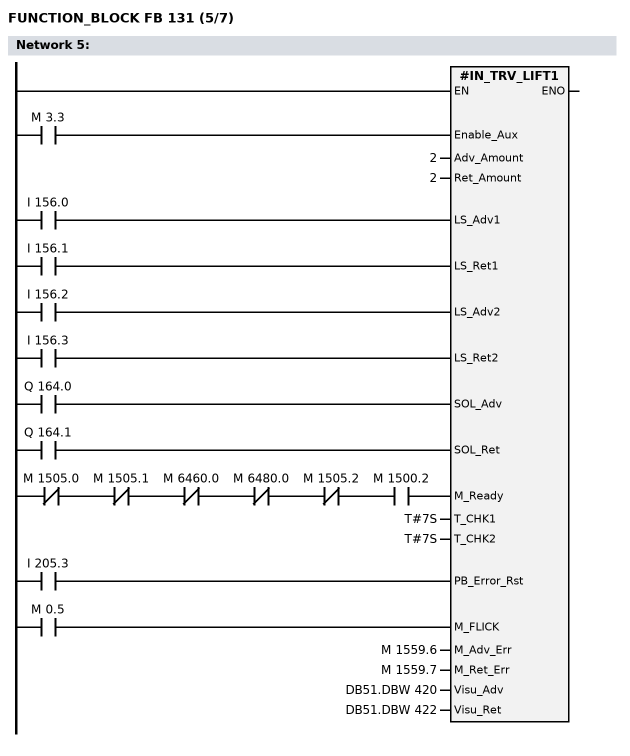

      A     M      3.3;
      =     L      0.0;
      BLD   103;
      A     I    156.0;
      =     L      0.1;
      BLD   103;
      A     I    156.1;
      =     L      0.2;
      BLD   103;
      A     I    156.2;
      =     L      0.3;
      BLD   103;
      A     I    156.3;
      =     L      0.4;
      BLD   103;
      A     Q    164.0;
      =     L      1.1;
      BLD   103;
      A     Q    164.1;
      =     L      1.2;
      BLD   103;
      AN    M   1505.0;
      AN    M   1505.1;
      AN    M   6460.0;
      AN    M   6480.0;
      AN    M   1505.2;
      A     M   1500.2;
      =     L      1.3;
      BLD   103;
      A     I    205.3;
      =     L      1.5;
      BLD   103;
      A     M      0.5;
      =     L      1.6;
      BLD   103;
      CALL #IN_TRV_LIFT1 (
           Enable_Aux               := L      0.0,
           Adv_Amount               := 2,
           Ret_Amount               := 2,
           LS_Adv1                  := L      0.1,
           LS_Ret1                  := L      0.2,
           LS_Adv2                  := L      0.3,
           LS_Ret2                  := L      0.4,
           SOL_Adv                  := L      1.1,
           SOL_Ret                  := L      1.2,
           M_Ready                  := L      1.3,
           T_CHK1                   := T#7S,
           T_CHK2                   := T#7S,
           PB_Error_Rst             := L      1.5,
           M_FLICK                  := L      1.6,
           M_Adv_Err                := M   1559.6,
           M_Ret_Err                := M   1559.7,
           Visu_Adv                 := DB51.DBW  420,
           Visu_Ret                 := DB51.DBW  422);
      NOP   0;
NETWORK
TITLE =
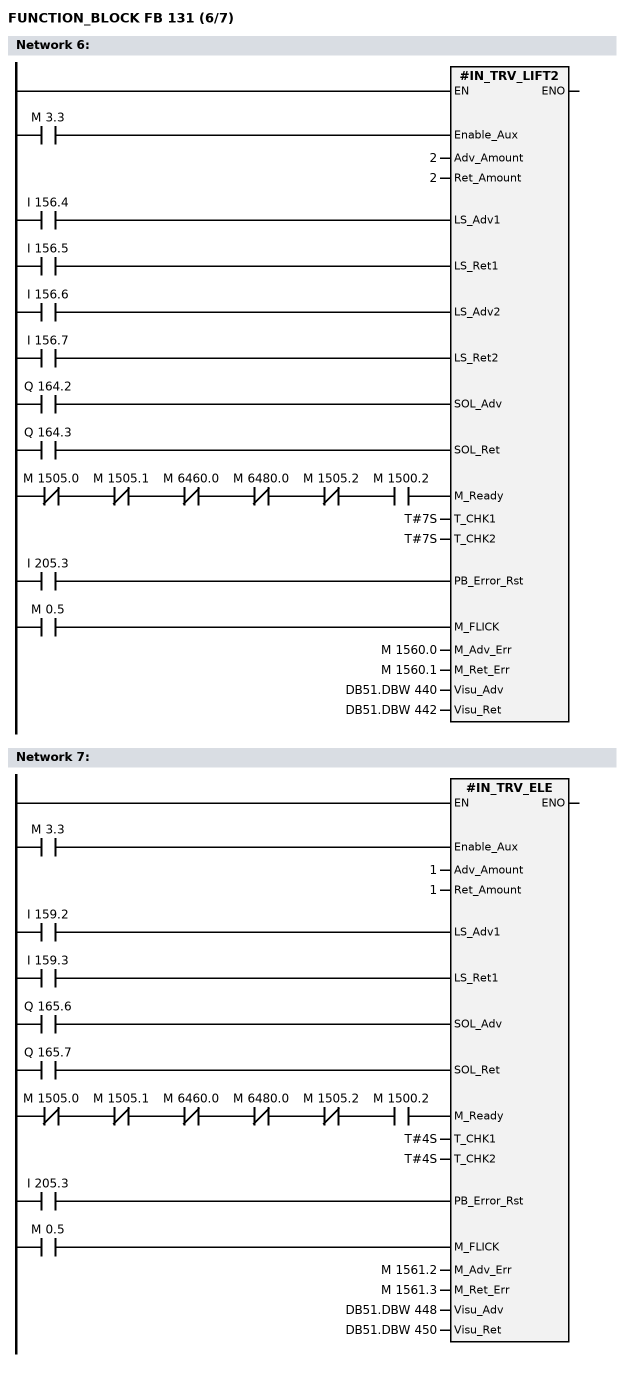

      A     M      3.3;
      =     L      0.0;
      BLD   103;
      A     I    156.4;
      =     L      0.1;
      BLD   103;
      A     I    156.5;
      =     L      0.2;
      BLD   103;
      A     I    156.6;
      =     L      0.3;
      BLD   103;
      A     I    156.7;
      =     L      0.4;
      BLD   103;
      A     Q    164.2;
      =     L      1.1;
      BLD   103;
      A     Q    164.3;
      =     L      1.2;
      BLD   103;
      AN    M   1505.0;
      AN    M   1505.1;
      AN    M   6460.0;
      AN    M   6480.0;
      AN    M   1505.2;
      A     M   1500.2;
      =     L      1.3;
      BLD   103;
      A     I    205.3;
      =     L      1.5;
      BLD   103;
      A     M      0.5;
      =     L      1.6;
      BLD   103;
      CALL #IN_TRV_LIFT2 (
           Enable_Aux               := L      0.0,
           Adv_Amount               := 2,
           Ret_Amount               := 2,
           LS_Adv1                  := L      0.1,
           LS_Ret1                  := L      0.2,
           LS_Adv2                  := L      0.3,
           LS_Ret2                  := L      0.4,
           SOL_Adv                  := L      1.1,
           SOL_Ret                  := L      1.2,
           M_Ready                  := L      1.3,
           T_CHK1                   := T#7S,
           T_CHK2                   := T#7S,
           PB_Error_Rst             := L      1.5,
           M_FLICK                  := L      1.6,
           M_Adv_Err                := M   1560.0,
           M_Ret_Err                := M   1560.1,
           Visu_Adv                 := DB51.DBW  440,
           Visu_Ret                 := DB51.DBW  442);
      NOP   0;
NETWORK
TITLE =

      A     M      3.3;
      =     L      0.0;
      BLD   103;
      A     I    159.2;
      =     L      0.1;
      BLD   103;
      A     I    159.3;
      =     L      0.2;
      BLD   103;
      A     Q    165.6;
      =     L      1.1;
      BLD   103;
      A     Q    165.7;
      =     L      1.2;
      BLD   103;
      AN    M   1505.0;
      AN    M   1505.1;
      AN    M   6460.0;
      AN    M   6480.0;
      AN    M   1505.2;
      A     M   1500.2;
      =     L      1.3;
      BLD   103;
      A     I    205.3;
      =     L      1.5;
      BLD   103;
      A     M      0.5;
      =     L      1.6;
      BLD   103;
      CALL #IN_TRV_ELE (
           Enable_Aux               := L      0.0,
           Adv_Amount               := 1,
           Ret_Amount               := 1,
           LS_Adv1                  := L      0.1,
           LS_Ret1                  := L      0.2,
           SOL_Adv                  := L      1.1,
           SOL_Ret                  := L      1.2,
           M_Ready                  := L      1.3,
           T_CHK1                   := T#4S,
           T_CHK2                   := T#4S,
           PB_Error_Rst             := L      1.5,
           M_FLICK                  := L      1.6,
           M_Adv_Err                := M   1561.2,
           M_Ret_Err                := M   1561.3,
           Visu_Adv                 := DB51.DBW  448,
           Visu_Ret                 := DB51.DBW  450);
      NOP   0;
NETWORK
TITLE =
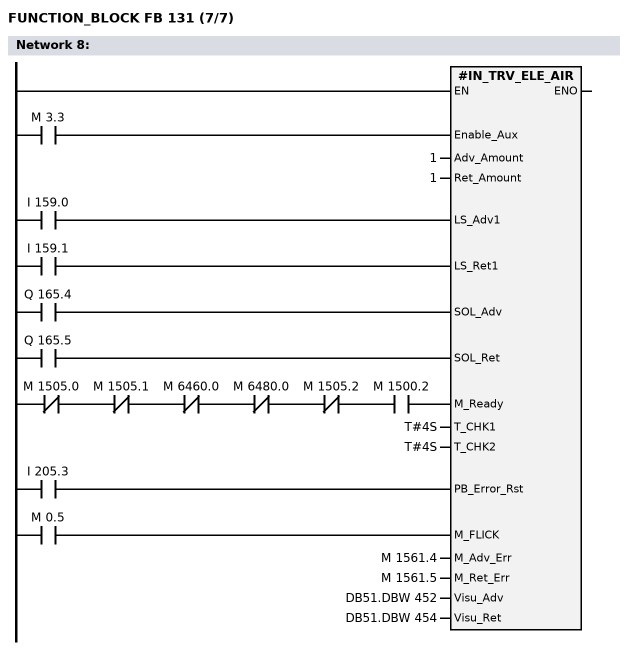

      A     M      3.3;
      =     L      0.0;
      BLD   103;
      A     I    159.0;
      =     L      0.1;
      BLD   103;
      A     I    159.1;
      =     L      0.2;
      BLD   103;
      A     Q    165.4;
      =     L      1.1;
      BLD   103;
      A     Q    165.5;
      =     L      1.2;
      BLD   103;
      AN    M   1505.0;
      AN    M   1505.1;
      AN    M   6460.0;
      AN    M   6480.0;
      AN    M   1505.2;
      A     M   1500.2;
      =     L      1.3;
      BLD   103;
      A     I    205.3;
      =     L      1.5;
      BLD   103;
      A     M      0.5;
      =     L      1.6;
      BLD   103;
      CALL #IN_TRV_ELE_AIR (
           Enable_Aux               := L      0.0,
           Adv_Amount               := 1,
           Ret_Amount               := 1,
           LS_Adv1                  := L      0.1,
           LS_Ret1                  := L      0.2,
           SOL_Adv                  := L      1.1,
           SOL_Ret                  := L      1.2,
           M_Ready                  := L      1.3,
           T_CHK1                   := T#4S,
           T_CHK2                   := T#4S,
           PB_Error_Rst             := L      1.5,
           M_FLICK                  := L      1.6,
           M_Adv_Err                := M   1561.4,
           M_Ret_Err                := M   1561.5,
           Visu_Adv                 := DB51.DBW  452,
           Visu_Ret                 := DB51.DBW  454);
      NOP   0;
END_FUNCTION_BLOCK

DATA_BLOCK DB 131
TITLE =
VERSION : 0.0

 FB 131
BEGIN
   IN_TRV_CUSHION_B.Enable_Aux := FALSE;
   IN_TRV_CUSHION_B.Adv_Amount := 0;
   IN_TRV_CUSHION_B.Ret_Amount := 0;
   IN_TRV_CUSHION_B.LS_Adv1 := FALSE;
   IN_TRV_CUSHION_B.LS_Ret1 := FALSE;
   IN_TRV_CUSHION_B.LS_Adv2 := FALSE;
   IN_TRV_CUSHION_B.LS_Ret2 := FALSE;
   IN_TRV_CUSHION_B.LS_Adv3 := FALSE;
   IN_TRV_CUSHION_B.LS_Ret3 := FALSE;
   IN_TRV_CUSHION_B.LS_Adv4 := FALSE;
   IN_TRV_CUSHION_B.LS_Ret4 := FALSE;
   IN_TRV_CUSHION_B.SOL_Adv := FALSE;
   IN_TRV_CUSHION_B.SOL_Ret := FALSE;
   IN_TRV_CUSHION_B.M_Ready := FALSE;
   IN_TRV_CUSHION_B.T_CHK1 := T#0MS;
   IN_TRV_CUSHION_B.T_CHK2 := T#0MS;
   IN_TRV_CUSHION_B.PB_Lamp_CHK := FALSE;
   IN_TRV_CUSHION_B.PB_Error_Rst := FALSE;
   IN_TRV_CUSHION_B.M_FLICK := FALSE;
   IN_TRV_CUSHION_B.M_Adv_Err := FALSE;
   IN_TRV_CUSHION_B.M_Ret_Err := FALSE;
   IN_TRV_CUSHION_B.LP_Adv := FALSE;
   IN_TRV_CUSHION_B.LP_Ret := FALSE;
   IN_TRV_CUSHION_B.Visu_Adv := W#16#0;
   IN_TRV_CUSHION_B.Visu_Ret := W#16#0;
   IN_TRV_CUSHION_B.Error_T1.IN := FALSE;
   IN_TRV_CUSHION_B.Error_T1.PT := T#0MS;
   IN_TRV_CUSHION_B.Error_T1.Q := FALSE;
   IN_TRV_CUSHION_B.Error_T1.ET := T#0MS;
   IN_TRV_CUSHION_B.Error_T1.STATE := B#16#0;
   IN_TRV_CUSHION_B.Error_T1.STIME := T#0MS;
   IN_TRV_CUSHION_B.Error_T1.ATIME := T#0MS;
   IN_TRV_CUSHION_B.Error_T2.IN := FALSE;
   IN_TRV_CUSHION_B.Error_T2.PT := T#0MS;
   IN_TRV_CUSHION_B.Error_T2.Q := FALSE;
   IN_TRV_CUSHION_B.Error_T2.ET := T#0MS;
   IN_TRV_CUSHION_B.Error_T2.STATE := B#16#0;
   IN_TRV_CUSHION_B.Error_T2.STIME := T#0MS;
   IN_TRV_CUSHION_B.Error_T2.ATIME := T#0MS;
   IN_TRV_CUSHION_B.CHK_Aux1 := FALSE;
   IN_TRV_CUSHION_B.CHK_Aux2 := FALSE;
   IN_TRV_CUSHION_B.Error_T1_DN := FALSE;
   IN_TRV_CUSHION_B.Error_T2_DN := FALSE;
   IN_TRV_CUSHION_B.Adv_Memo := FALSE;
   IN_TRV_CUSHION_B.Visu_Adv_Arr[0] := FALSE;
   IN_TRV_CUSHION_B.Visu_Adv_Arr[1] := FALSE;
   IN_TRV_CUSHION_B.Visu_Adv_Arr[2] := FALSE;
   IN_TRV_CUSHION_B.Visu_Adv_Arr[3] := FALSE;
   IN_TRV_CUSHION_B.Visu_Adv_Arr[4] := FALSE;
   IN_TRV_CUSHION_B.Visu_Adv_Arr[5] := FALSE;
   IN_TRV_CUSHION_B.Visu_Adv_Arr[6] := FALSE;
   IN_TRV_CUSHION_B.Visu_Adv_Arr[7] := FALSE;
   IN_TRV_CUSHION_B.Visu_Adv_Arr[8] := FALSE;
   IN_TRV_CUSHION_B.Visu_Adv_Arr[9] := FALSE;
   IN_TRV_CUSHION_B.Visu_Adv_Arr[10] := FALSE;
   IN_TRV_CUSHION_B.Visu_Adv_Arr[11] := FALSE;
   IN_TRV_CUSHION_B.Visu_Adv_Arr[12] := FALSE;
   IN_TRV_CUSHION_B.Visu_Adv_Arr[13] := FALSE;
   IN_TRV_CUSHION_B.Visu_Adv_Arr[14] := FALSE;
   IN_TRV_CUSHION_B.Visu_Adv_Arr[15] := FALSE;
   IN_TRV_CUSHION_B.Visu_Ret_Arr[0] := FALSE;
   IN_TRV_CUSHION_B.Visu_Ret_Arr[1] := FALSE;
   IN_TRV_CUSHION_B.Visu_Ret_Arr[2] := FALSE;
   IN_TRV_CUSHION_B.Visu_Ret_Arr[3] := FALSE;
   IN_TRV_CUSHION_B.Visu_Ret_Arr[4] := FALSE;
   IN_TRV_CUSHION_B.Visu_Ret_Arr[5] := FALSE;
   IN_TRV_CUSHION_B.Visu_Ret_Arr[6] := FALSE;
   IN_TRV_CUSHION_B.Visu_Ret_Arr[7] := FALSE;
   IN_TRV_CUSHION_B.Visu_Ret_Arr[8] := FALSE;
   IN_TRV_CUSHION_B.Visu_Ret_Arr[9] := FALSE;
   IN_TRV_CUSHION_B.Visu_Ret_Arr[10] := FALSE;
   IN_TRV_CUSHION_B.Visu_Ret_Arr[11] := FALSE;
   IN_TRV_CUSHION_B.Visu_Ret_Arr[12] := FALSE;
   IN_TRV_CUSHION_B.Visu_Ret_Arr[13] := FALSE;
   IN_TRV_CUSHION_B.Visu_Ret_Arr[14] := FALSE;
   IN_TRV_CUSHION_B.Visu_Ret_Arr[15] := FALSE;
   IN_TRV_CUSHION_B.BLK_Move_Ret := 0;
   IN_TRV_CUSHION_B.Enable := FALSE;
   IN_TRV_CUSHION_B.Adv_End := FALSE;
   IN_TRV_CUSHION_B.Ret_End := FALSE;
   IN_TRV_GUIDE.Enable_Aux := FALSE;
   IN_TRV_GUIDE.Adv_Amount := 0;
   IN_TRV_GUIDE.Ret_Amount := 0;
   IN_TRV_GUIDE.LS_Adv1 := FALSE;
   IN_TRV_GUIDE.LS_Ret1 := FALSE;
   IN_TRV_GUIDE.LS_Adv2 := FALSE;
   IN_TRV_GUIDE.LS_Ret2 := FALSE;
   IN_TRV_GUIDE.LS_Adv3 := FALSE;
   IN_TRV_GUIDE.LS_Ret3 := FALSE;
   IN_TRV_GUIDE.LS_Adv4 := FALSE;
   IN_TRV_GUIDE.LS_Ret4 := FALSE;
   IN_TRV_GUIDE.SOL_Adv := FALSE;
   IN_TRV_GUIDE.SOL_Ret := FALSE;
   IN_TRV_GUIDE.M_Ready := FALSE;
   IN_TRV_GUIDE.T_CHK1 := T#0MS;
   IN_TRV_GUIDE.T_CHK2 := T#0MS;
   IN_TRV_GUIDE.PB_Lamp_CHK := FALSE;
   IN_TRV_GUIDE.PB_Error_Rst := FALSE;
   IN_TRV_GUIDE.M_FLICK := FALSE;
   IN_TRV_GUIDE.M_Adv_Err := FALSE;
   IN_TRV_GUIDE.M_Ret_Err := FALSE;
   IN_TRV_GUIDE.LP_Adv := FALSE;
   IN_TRV_GUIDE.LP_Ret := FALSE;
   IN_TRV_GUIDE.Visu_Adv := W#16#0;
   IN_TRV_GUIDE.Visu_Ret := W#16#0;
   IN_TRV_GUIDE.Error_T1.IN := FALSE;
   IN_TRV_GUIDE.Error_T1.PT := T#0MS;
   IN_TRV_GUIDE.Error_T1.Q := FALSE;
   IN_TRV_GUIDE.Error_T1.ET := T#0MS;
   IN_TRV_GUIDE.Error_T1.STATE := B#16#0;
   IN_TRV_GUIDE.Error_T1.STIME := T#0MS;
   IN_TRV_GUIDE.Error_T1.ATIME := T#0MS;
   IN_TRV_GUIDE.Error_T2.IN := FALSE;
   IN_TRV_GUIDE.Error_T2.PT := T#0MS;
   IN_TRV_GUIDE.Error_T2.Q := FALSE;
   IN_TRV_GUIDE.Error_T2.ET := T#0MS;
   IN_TRV_GUIDE.Error_T2.STATE := B#16#0;
   IN_TRV_GUIDE.Error_T2.STIME := T#0MS;
   IN_TRV_GUIDE.Error_T2.ATIME := T#0MS;
   IN_TRV_GUIDE.CHK_Aux1 := FALSE;
   IN_TRV_GUIDE.CHK_Aux2 := FALSE;
   IN_TRV_GUIDE.Error_T1_DN := FALSE;
   IN_TRV_GUIDE.Error_T2_DN := FALSE;
   IN_TRV_GUIDE.Adv_Memo := FALSE;
   IN_TRV_GUIDE.Visu_Adv_Arr[0] := FALSE;
   IN_TRV_GUIDE.Visu_Adv_Arr[1] := FALSE;
   IN_TRV_GUIDE.Visu_Adv_Arr[2] := FALSE;
   IN_TRV_GUIDE.Visu_Adv_Arr[3] := FALSE;
   IN_TRV_GUIDE.Visu_Adv_Arr[4] := FALSE;
   IN_TRV_GUIDE.Visu_Adv_Arr[5] := FALSE;
   IN_TRV_GUIDE.Visu_Adv_Arr[6] := FALSE;
   IN_TRV_GUIDE.Visu_Adv_Arr[7] := FALSE;
   IN_TRV_GUIDE.Visu_Adv_Arr[8] := FALSE;
   IN_TRV_GUIDE.Visu_Adv_Arr[9] := FALSE;
   IN_TRV_GUIDE.Visu_Adv_Arr[10] := FALSE;
   IN_TRV_GUIDE.Visu_Adv_Arr[11] := FALSE;
   IN_TRV_GUIDE.Visu_Adv_Arr[12] := FALSE;
   IN_TRV_GUIDE.Visu_Adv_Arr[13] := FALSE;
   IN_TRV_GUIDE.Visu_Adv_Arr[14] := FALSE;
   IN_TRV_GUIDE.Visu_Adv_Arr[15] := FALSE;
   IN_TRV_GUIDE.Visu_Ret_Arr[0] := FALSE;
   IN_TRV_GUIDE.Visu_Ret_Arr[1] := FALSE;
   IN_TRV_GUIDE.Visu_Ret_Arr[2] := FALSE;
   IN_TRV_GUIDE.Visu_Ret_Arr[3] := FALSE;
   IN_TRV_GUIDE.Visu_Ret_Arr[4] := FALSE;
   IN_TRV_GUIDE.Visu_Ret_Arr[5] := FALSE;
   IN_TRV_GUIDE.Visu_Ret_Arr[6] := FALSE;
   IN_TRV_GUIDE.Visu_Ret_Arr[7] := FALSE;
   IN_TRV_GUIDE.Visu_Ret_Arr[8] := FALSE;
   IN_TRV_GUIDE.Visu_Ret_Arr[9] := FALSE;
   IN_TRV_GUIDE.Visu_Ret_Arr[10] := FALSE;
   IN_TRV_GUIDE.Visu_Ret_Arr[11] := FALSE;
   IN_TRV_GUIDE.Visu_Ret_Arr[12] := FALSE;
   IN_TRV_GUIDE.Visu_Ret_Arr[13] := FALSE;
   IN_TRV_GUIDE.Visu_Ret_Arr[14] := FALSE;
   IN_TRV_GUIDE.Visu_Ret_Arr[15] := FALSE;
   IN_TRV_GUIDE.BLK_Move_Ret := 0;
   IN_TRV_GUIDE.Enable := FALSE;
   IN_TRV_GUIDE.Adv_End := FALSE;
   IN_TRV_GUIDE.Ret_End := FALSE;
   IN_TRV_CLAMP.Enable_Aux := FALSE;
   IN_TRV_CLAMP.Adv_Amount := 0;
   IN_TRV_CLAMP.Ret_Amount := 0;
   IN_TRV_CLAMP.LS_Adv1 := FALSE;
   IN_TRV_CLAMP.LS_Ret1 := FALSE;
   IN_TRV_CLAMP.LS_Adv2 := FALSE;
   IN_TRV_CLAMP.LS_Ret2 := FALSE;
   IN_TRV_CLAMP.LS_Adv3 := FALSE;
   IN_TRV_CLAMP.LS_Ret3 := FALSE;
   IN_TRV_CLAMP.LS_Adv4 := FALSE;
   IN_TRV_CLAMP.LS_Ret4 := FALSE;
   IN_TRV_CLAMP.SOL_Adv := FALSE;
   IN_TRV_CLAMP.SOL_Ret := FALSE;
   IN_TRV_CLAMP.M_Ready := FALSE;
   IN_TRV_CLAMP.T_CHK1 := T#0MS;
   IN_TRV_CLAMP.T_CHK2 := T#0MS;
   IN_TRV_CLAMP.PB_Lamp_CHK := FALSE;
   IN_TRV_CLAMP.PB_Error_Rst := FALSE;
   IN_TRV_CLAMP.M_FLICK := FALSE;
   IN_TRV_CLAMP.M_Adv_Err := FALSE;
   IN_TRV_CLAMP.M_Ret_Err := FALSE;
   IN_TRV_CLAMP.LP_Adv := FALSE;
   IN_TRV_CLAMP.LP_Ret := FALSE;
   IN_TRV_CLAMP.Visu_Adv := W#16#0;
   IN_TRV_CLAMP.Visu_Ret := W#16#0;
   IN_TRV_CLAMP.Error_T1.IN := FALSE;
   IN_TRV_CLAMP.Error_T1.PT := T#0MS;
   IN_TRV_CLAMP.Error_T1.Q := FALSE;
   IN_TRV_CLAMP.Error_T1.ET := T#0MS;
   IN_TRV_CLAMP.Error_T1.STATE := B#16#0;
   IN_TRV_CLAMP.Error_T1.STIME := T#0MS;
   IN_TRV_CLAMP.Error_T1.ATIME := T#0MS;
   IN_TRV_CLAMP.Error_T2.IN := FALSE;
   IN_TRV_CLAMP.Error_T2.PT := T#0MS;
   IN_TRV_CLAMP.Error_T2.Q := FALSE;
   IN_TRV_CLAMP.Error_T2.ET := T#0MS;
   IN_TRV_CLAMP.Error_T2.STATE := B#16#0;
   IN_TRV_CLAMP.Error_T2.STIME := T#0MS;
   IN_TRV_CLAMP.Error_T2.ATIME := T#0MS;
   IN_TRV_CLAMP.CHK_Aux1 := FALSE;
   IN_TRV_CLAMP.CHK_Aux2 := FALSE;
   IN_TRV_CLAMP.Error_T1_DN := FALSE;
   IN_TRV_CLAMP.Error_T2_DN := FALSE;
   IN_TRV_CLAMP.Adv_Memo := FALSE;
   IN_TRV_CLAMP.Visu_Adv_Arr[0] := FALSE;
   IN_TRV_CLAMP.Visu_Adv_Arr[1] := FALSE;
   IN_TRV_CLAMP.Visu_Adv_Arr[2] := FALSE;
   IN_TRV_CLAMP.Visu_Adv_Arr[3] := FALSE;
   IN_TRV_CLAMP.Visu_Adv_Arr[4] := FALSE;
   IN_TRV_CLAMP.Visu_Adv_Arr[5] := FALSE;
   IN_TRV_CLAMP.Visu_Adv_Arr[6] := FALSE;
   IN_TRV_CLAMP.Visu_Adv_Arr[7] := FALSE;
   IN_TRV_CLAMP.Visu_Adv_Arr[8] := FALSE;
   IN_TRV_CLAMP.Visu_Adv_Arr[9] := FALSE;
   IN_TRV_CLAMP.Visu_Adv_Arr[10] := FALSE;
   IN_TRV_CLAMP.Visu_Adv_Arr[11] := FALSE;
   IN_TRV_CLAMP.Visu_Adv_Arr[12] := FALSE;
   IN_TRV_CLAMP.Visu_Adv_Arr[13] := FALSE;
   IN_TRV_CLAMP.Visu_Adv_Arr[14] := FALSE;
   IN_TRV_CLAMP.Visu_Adv_Arr[15] := FALSE;
   IN_TRV_CLAMP.Visu_Ret_Arr[0] := FALSE;
   IN_TRV_CLAMP.Visu_Ret_Arr[1] := FALSE;
   IN_TRV_CLAMP.Visu_Ret_Arr[2] := FALSE;
   IN_TRV_CLAMP.Visu_Ret_Arr[3] := FALSE;
   IN_TRV_CLAMP.Visu_Ret_Arr[4] := FALSE;
   IN_TRV_CLAMP.Visu_Ret_Arr[5] := FALSE;
   IN_TRV_CLAMP.Visu_Ret_Arr[6] := FALSE;
   IN_TRV_CLAMP.Visu_Ret_Arr[7] := FALSE;
   IN_TRV_CLAMP.Visu_Ret_Arr[8] := FALSE;
   IN_TRV_CLAMP.Visu_Ret_Arr[9] := FALSE;
   IN_TRV_CLAMP.Visu_Ret_Arr[10] := FALSE;
   IN_TRV_CLAMP.Visu_Ret_Arr[11] := FALSE;
   IN_TRV_CLAMP.Visu_Ret_Arr[12] := FALSE;
   IN_TRV_CLAMP.Visu_Ret_Arr[13] := FALSE;
   IN_TRV_CLAMP.Visu_Ret_Arr[14] := FALSE;
   IN_TRV_CLAMP.Visu_Ret_Arr[15] := FALSE;
   IN_TRV_CLAMP.BLK_Move_Ret := 0;
   IN_TRV_CLAMP.Enable := FALSE;
   IN_TRV_CLAMP.Adv_End := FALSE;
   IN_TRV_CLAMP.Ret_End := FALSE;
   IN_TRV_STOPPER.Enable_Aux := FALSE;
   IN_TRV_STOPPER.Adv_Amount := 0;
   IN_TRV_STOPPER.Ret_Amount := 0;
   IN_TRV_STOPPER.LS_Adv1 := FALSE;
   IN_TRV_STOPPER.LS_Ret1 := FALSE;
   IN_TRV_STOPPER.LS_Adv2 := FALSE;
   IN_TRV_STOPPER.LS_Ret2 := FALSE;
   IN_TRV_STOPPER.LS_Adv3 := FALSE;
   IN_TRV_STOPPER.LS_Ret3 := FALSE;
   IN_TRV_STOPPER.LS_Adv4 := FALSE;
   IN_TRV_STOPPER.LS_Ret4 := FALSE;
   IN_TRV_STOPPER.SOL_Adv := FALSE;
   IN_TRV_STOPPER.SOL_Ret := FALSE;
   IN_TRV_STOPPER.M_Ready := FALSE;
   IN_TRV_STOPPER.T_CHK1 := T#0MS;
   IN_TRV_STOPPER.T_CHK2 := T#0MS;
   IN_TRV_STOPPER.PB_Lamp_CHK := FALSE;
   IN_TRV_STOPPER.PB_Error_Rst := FALSE;
   IN_TRV_STOPPER.M_FLICK := FALSE;
   IN_TRV_STOPPER.M_Adv_Err := FALSE;
   IN_TRV_STOPPER.M_Ret_Err := FALSE;
   IN_TRV_STOPPER.LP_Adv := FALSE;
   IN_TRV_STOPPER.LP_Ret := FALSE;
   IN_TRV_STOPPER.Visu_Adv := W#16#0;
   IN_TRV_STOPPER.Visu_Ret := W#16#0;
   IN_TRV_STOPPER.Error_T1.IN := FALSE;
   IN_TRV_STOPPER.Error_T1.PT := T#0MS;
   IN_TRV_STOPPER.Error_T1.Q := FALSE;
   IN_TRV_STOPPER.Error_T1.ET := T#0MS;
   IN_TRV_STOPPER.Error_T1.STATE := B#16#0;
   IN_TRV_STOPPER.Error_T1.STIME := T#0MS;
   IN_TRV_STOPPER.Error_T1.ATIME := T#0MS;
   IN_TRV_STOPPER.Error_T2.IN := FALSE;
   IN_TRV_STOPPER.Error_T2.PT := T#0MS;
   IN_TRV_STOPPER.Error_T2.Q := FALSE;
   IN_TRV_STOPPER.Error_T2.ET := T#0MS;
   IN_TRV_STOPPER.Error_T2.STATE := B#16#0;
   IN_TRV_STOPPER.Error_T2.STIME := T#0MS;
   IN_TRV_STOPPER.Error_T2.ATIME := T#0MS;
   IN_TRV_STOPPER.CHK_Aux1 := FALSE;
   IN_TRV_STOPPER.CHK_Aux2 := FALSE;
   IN_TRV_STOPPER.Error_T1_DN := FALSE;
   IN_TRV_STOPPER.Error_T2_DN := FALSE;
   IN_TRV_STOPPER.Adv_Memo := FALSE;
   IN_TRV_STOPPER.Visu_Adv_Arr[0] := FALSE;
   IN_TRV_STOPPER.Visu_Adv_Arr[1] := FALSE;
   IN_TRV_STOPPER.Visu_Adv_Arr[2] := FALSE;
   IN_TRV_STOPPER.Visu_Adv_Arr[3] := FALSE;
   IN_TRV_STOPPER.Visu_Adv_Arr[4] := FALSE;
   IN_TRV_STOPPER.Visu_Adv_Arr[5] := FALSE;
   IN_TRV_STOPPER.Visu_Adv_Arr[6] := FALSE;
   IN_TRV_STOPPER.Visu_Adv_Arr[7] := FALSE;
   IN_TRV_STOPPER.Visu_Adv_Arr[8] := FALSE;
   IN_TRV_STOPPER.Visu_Adv_Arr[9] := FALSE;
   IN_TRV_STOPPER.Visu_Adv_Arr[10] := FALSE;
   IN_TRV_STOPPER.Visu_Adv_Arr[11] := FALSE;
   IN_TRV_STOPPER.Visu_Adv_Arr[12] := FALSE;
   IN_TRV_STOPPER.Visu_Adv_Arr[13] := FALSE;
   IN_TRV_STOPPER.Visu_Adv_Arr[14] := FALSE;
   IN_TRV_STOPPER.Visu_Adv_Arr[15] := FALSE;
   IN_TRV_STOPPER.Visu_Ret_Arr[0] := FALSE;
   IN_TRV_STOPPER.Visu_Ret_Arr[1] := FALSE;
   IN_TRV_STOPPER.Visu_Ret_Arr[2] := FALSE;
   IN_TRV_STOPPER.Visu_Ret_Arr[3] := FALSE;
   IN_TRV_STOPPER.Visu_Ret_Arr[4] := FALSE;
   IN_TRV_STOPPER.Visu_Ret_Arr[5] := FALSE;
   IN_TRV_STOPPER.Visu_Ret_Arr[6] := FALSE;
   IN_TRV_STOPPER.Visu_Ret_Arr[7] := FALSE;
   IN_TRV_STOPPER.Visu_Ret_Arr[8] := FALSE;
   IN_TRV_STOPPER.Visu_Ret_Arr[9] := FALSE;
   IN_TRV_STOPPER.Visu_Ret_Arr[10] := FALSE;
   IN_TRV_STOPPER.Visu_Ret_Arr[11] := FALSE;
   IN_TRV_STOPPER.Visu_Ret_Arr[12] := FALSE;
   IN_TRV_STOPPER.Visu_Ret_Arr[13] := FALSE;
   IN_TRV_STOPPER.Visu_Ret_Arr[14] := FALSE;
   IN_TRV_STOPPER.Visu_Ret_Arr[15] := FALSE;
   IN_TRV_STOPPER.BLK_Move_Ret := 0;
   IN_TRV_STOPPER.Enable := FALSE;
   IN_TRV_STOPPER.Adv_End := FALSE;
   IN_TRV_STOPPER.Ret_End := FALSE;
   IN_TRV_LIFT1.Enable_Aux := FALSE;
   IN_TRV_LIFT1.Adv_Amount := 0;
   IN_TRV_LIFT1.Ret_Amount := 0;
   IN_TRV_LIFT1.LS_Adv1 := FALSE;
   IN_TRV_LIFT1.LS_Ret1 := FALSE;
   IN_TRV_LIFT1.LS_Adv2 := FALSE;
   IN_TRV_LIFT1.LS_Ret2 := FALSE;
   IN_TRV_LIFT1.LS_Adv3 := FALSE;
   IN_TRV_LIFT1.LS_Ret3 := FALSE;
   IN_TRV_LIFT1.LS_Adv4 := FALSE;
   IN_TRV_LIFT1.LS_Ret4 := FALSE;
   IN_TRV_LIFT1.SOL_Adv := FALSE;
   IN_TRV_LIFT1.SOL_Ret := FALSE;
   IN_TRV_LIFT1.M_Ready := FALSE;
   IN_TRV_LIFT1.T_CHK1 := T#0MS;
   IN_TRV_LIFT1.T_CHK2 := T#0MS;
   IN_TRV_LIFT1.PB_Lamp_CHK := FALSE;
   IN_TRV_LIFT1.PB_Error_Rst := FALSE;
   IN_TRV_LIFT1.M_FLICK := FALSE;
   IN_TRV_LIFT1.M_Adv_Err := FALSE;
   IN_TRV_LIFT1.M_Ret_Err := FALSE;
   IN_TRV_LIFT1.LP_Adv := FALSE;
   IN_TRV_LIFT1.LP_Ret := FALSE;
   IN_TRV_LIFT1.Visu_Adv := W#16#0;
   IN_TRV_LIFT1.Visu_Ret := W#16#0;
   IN_TRV_LIFT1.Error_T1.IN := FALSE;
   IN_TRV_LIFT1.Error_T1.PT := T#0MS;
   IN_TRV_LIFT1.Error_T1.Q := FALSE;
   IN_TRV_LIFT1.Error_T1.ET := T#0MS;
   IN_TRV_LIFT1.Error_T1.STATE := B#16#0;
   IN_TRV_LIFT1.Error_T1.STIME := T#0MS;
   IN_TRV_LIFT1.Error_T1.ATIME := T#0MS;
   IN_TRV_LIFT1.Error_T2.IN := FALSE;
   IN_TRV_LIFT1.Error_T2.PT := T#0MS;
   IN_TRV_LIFT1.Error_T2.Q := FALSE;
   IN_TRV_LIFT1.Error_T2.ET := T#0MS;
   IN_TRV_LIFT1.Error_T2.STATE := B#16#0;
   IN_TRV_LIFT1.Error_T2.STIME := T#0MS;
   IN_TRV_LIFT1.Error_T2.ATIME := T#0MS;
   IN_TRV_LIFT1.CHK_Aux1 := FALSE;
   IN_TRV_LIFT1.CHK_Aux2 := FALSE;
   IN_TRV_LIFT1.Error_T1_DN := FALSE;
   IN_TRV_LIFT1.Error_T2_DN := FALSE;
   IN_TRV_LIFT1.Adv_Memo := FALSE;
   IN_TRV_LIFT1.Visu_Adv_Arr[0] := FALSE;
   IN_TRV_LIFT1.Visu_Adv_Arr[1] := FALSE;
   IN_TRV_LIFT1.Visu_Adv_Arr[2] := FALSE;
   IN_TRV_LIFT1.Visu_Adv_Arr[3] := FALSE;
   IN_TRV_LIFT1.Visu_Adv_Arr[4] := FALSE;
   IN_TRV_LIFT1.Visu_Adv_Arr[5] := FALSE;
   IN_TRV_LIFT1.Visu_Adv_Arr[6] := FALSE;
   IN_TRV_LIFT1.Visu_Adv_Arr[7] := FALSE;
   IN_TRV_LIFT1.Visu_Adv_Arr[8] := FALSE;
   IN_TRV_LIFT1.Visu_Adv_Arr[9] := FALSE;
   IN_TRV_LIFT1.Visu_Adv_Arr[10] := FALSE;
   IN_TRV_LIFT1.Visu_Adv_Arr[11] := FALSE;
   IN_TRV_LIFT1.Visu_Adv_Arr[12] := FALSE;
   IN_TRV_LIFT1.Visu_Adv_Arr[13] := FALSE;
   IN_TRV_LIFT1.Visu_Adv_Arr[14] := FALSE;
   IN_TRV_LIFT1.Visu_Adv_Arr[15] := FALSE;
   IN_TRV_LIFT1.Visu_Ret_Arr[0] := FALSE;
   IN_TRV_LIFT1.Visu_Ret_Arr[1] := FALSE;
   IN_TRV_LIFT1.Visu_Ret_Arr[2] := FALSE;
   IN_TRV_LIFT1.Visu_Ret_Arr[3] := FALSE;
   IN_TRV_LIFT1.Visu_Ret_Arr[4] := FALSE;
   IN_TRV_LIFT1.Visu_Ret_Arr[5] := FALSE;
   IN_TRV_LIFT1.Visu_Ret_Arr[6] := FALSE;
   IN_TRV_LIFT1.Visu_Ret_Arr[7] := FALSE;
   IN_TRV_LIFT1.Visu_Ret_Arr[8] := FALSE;
   IN_TRV_LIFT1.Visu_Ret_Arr[9] := FALSE;
   IN_TRV_LIFT1.Visu_Ret_Arr[10] := FALSE;
   IN_TRV_LIFT1.Visu_Ret_Arr[11] := FALSE;
   IN_TRV_LIFT1.Visu_Ret_Arr[12] := FALSE;
   IN_TRV_LIFT1.Visu_Ret_Arr[13] := FALSE;
   IN_TRV_LIFT1.Visu_Ret_Arr[14] := FALSE;
   IN_TRV_LIFT1.Visu_Ret_Arr[15] := FALSE;
   IN_TRV_LIFT1.BLK_Move_Ret := 0;
   IN_TRV_LIFT1.Enable := FALSE;
   IN_TRV_LIFT1.Adv_End := FALSE;
   IN_TRV_LIFT1.Ret_End := FALSE;
   IN_TRV_ELE.Enable_Aux := FALSE;
   IN_TRV_ELE.Adv_Amount := 0;
   IN_TRV_ELE.Ret_Amount := 0;
   IN_TRV_ELE.LS_Adv1 := FALSE;
   IN_TRV_ELE.LS_Ret1 := FALSE;
   IN_TRV_ELE.LS_Adv2 := FALSE;
   IN_TRV_ELE.LS_Ret2 := FALSE;
   IN_TRV_ELE.LS_Adv3 := FALSE;
   IN_TRV_ELE.LS_Ret3 := FALSE;
   IN_TRV_ELE.LS_Adv4 := FALSE;
   IN_TRV_ELE.LS_Ret4 := FALSE;
   IN_TRV_ELE.SOL_Adv := FALSE;
   IN_TRV_ELE.SOL_Ret := FALSE;
   IN_TRV_ELE.M_Ready := FALSE;
   IN_TRV_ELE.T_CHK1 := T#0MS;
   IN_TRV_ELE.T_CHK2 := T#0MS;
   IN_TRV_ELE.PB_Lamp_CHK := FALSE;
   IN_TRV_ELE.PB_Error_Rst := FALSE;
   IN_TRV_ELE.M_FLICK := FALSE;
   IN_TRV_ELE.M_Adv_Err := FALSE;
   IN_TRV_ELE.M_Ret_Err := FALSE;
   IN_TRV_ELE.LP_Adv := FALSE;
   IN_TRV_ELE.LP_Ret := FALSE;
   IN_TRV_ELE.Visu_Adv := W#16#0;
   IN_TRV_ELE.Visu_Ret := W#16#0;
   IN_TRV_ELE.Error_T1.IN := FALSE;
   IN_TRV_ELE.Error_T1.PT := T#0MS;
   IN_TRV_ELE.Error_T1.Q := FALSE;
   IN_TRV_ELE.Error_T1.ET := T#0MS;
   IN_TRV_ELE.Error_T1.STATE := B#16#0;
   IN_TRV_ELE.Error_T1.STIME := T#0MS;
   IN_TRV_ELE.Error_T1.ATIME := T#0MS;
   IN_TRV_ELE.Error_T2.IN := FALSE;
   IN_TRV_ELE.Error_T2.PT := T#0MS;
   IN_TRV_ELE.Error_T2.Q := FALSE;
   IN_TRV_ELE.Error_T2.ET := T#0MS;
   IN_TRV_ELE.Error_T2.STATE := B#16#0;
   IN_TRV_ELE.Error_T2.STIME := T#0MS;
   IN_TRV_ELE.Error_T2.ATIME := T#0MS;
   IN_TRV_ELE.CHK_Aux1 := FALSE;
   IN_TRV_ELE.CHK_Aux2 := FALSE;
   IN_TRV_ELE.Error_T1_DN := FALSE;
   IN_TRV_ELE.Error_T2_DN := FALSE;
   IN_TRV_ELE.Adv_Memo := FALSE;
   IN_TRV_ELE.Visu_Adv_Arr[0] := FALSE;
   IN_TRV_ELE.Visu_Adv_Arr[1] := FALSE;
   IN_TRV_ELE.Visu_Adv_Arr[2] := FALSE;
   IN_TRV_ELE.Visu_Adv_Arr[3] := FALSE;
   IN_TRV_ELE.Visu_Adv_Arr[4] := FALSE;
   IN_TRV_ELE.Visu_Adv_Arr[5] := FALSE;
   IN_TRV_ELE.Visu_Adv_Arr[6] := FALSE;
   IN_TRV_ELE.Visu_Adv_Arr[7] := FALSE;
   IN_TRV_ELE.Visu_Adv_Arr[8] := FALSE;
   IN_TRV_ELE.Visu_Adv_Arr[9] := FALSE;
   IN_TRV_ELE.Visu_Adv_Arr[10] := FALSE;
   IN_TRV_ELE.Visu_Adv_Arr[11] := FALSE;
   IN_TRV_ELE.Visu_Adv_Arr[12] := FALSE;
   IN_TRV_ELE.Visu_Adv_Arr[13] := FALSE;
   IN_TRV_ELE.Visu_Adv_Arr[14] := FALSE;
   IN_TRV_ELE.Visu_Adv_Arr[15] := FALSE;
   IN_TRV_ELE.Visu_Ret_Arr[0] := FALSE;
   IN_TRV_ELE.Visu_Ret_Arr[1] := FALSE;
   IN_TRV_ELE.Visu_Ret_Arr[2] := FALSE;
   IN_TRV_ELE.Visu_Ret_Arr[3] := FALSE;
   IN_TRV_ELE.Visu_Ret_Arr[4] := FALSE;
   IN_TRV_ELE.Visu_Ret_Arr[5] := FALSE;
   IN_TRV_ELE.Visu_Ret_Arr[6] := FALSE;
   IN_TRV_ELE.Visu_Ret_Arr[7] := FALSE;
   IN_TRV_ELE.Visu_Ret_Arr[8] := FALSE;
   IN_TRV_ELE.Visu_Ret_Arr[9] := FALSE;
   IN_TRV_ELE.Visu_Ret_Arr[10] := FALSE;
   IN_TRV_ELE.Visu_Ret_Arr[11] := FALSE;
   IN_TRV_ELE.Visu_Ret_Arr[12] := FALSE;
   IN_TRV_ELE.Visu_Ret_Arr[13] := FALSE;
   IN_TRV_ELE.Visu_Ret_Arr[14] := FALSE;
   IN_TRV_ELE.Visu_Ret_Arr[15] := FALSE;
   IN_TRV_ELE.BLK_Move_Ret := 0;
   IN_TRV_ELE.Enable := FALSE;
   IN_TRV_ELE.Adv_End := FALSE;
   IN_TRV_ELE.Ret_End := FALSE;
   IN_TRV_LIFT2.Enable_Aux := FALSE;
   IN_TRV_LIFT2.Adv_Amount := 0;
   IN_TRV_LIFT2.Ret_Amount := 0;
   IN_TRV_LIFT2.LS_Adv1 := FALSE;
   IN_TRV_LIFT2.LS_Ret1 := FALSE;
   IN_TRV_LIFT2.LS_Adv2 := FALSE;
   IN_TRV_LIFT2.LS_Ret2 := FALSE;
   IN_TRV_LIFT2.LS_Adv3 := FALSE;
   IN_TRV_LIFT2.LS_Ret3 := FALSE;
   IN_TRV_LIFT2.LS_Adv4 := FALSE;
   IN_TRV_LIFT2.LS_Ret4 := FALSE;
   IN_TRV_LIFT2.SOL_Adv := FALSE;
   IN_TRV_LIFT2.SOL_Ret := FALSE;
   IN_TRV_LIFT2.M_Ready := FALSE;
   IN_TRV_LIFT2.T_CHK1 := T#0MS;
   IN_TRV_LIFT2.T_CHK2 := T#0MS;
   IN_TRV_LIFT2.PB_Lamp_CHK := FALSE;
   IN_TRV_LIFT2.PB_Error_Rst := FALSE;
   IN_TRV_LIFT2.M_FLICK := FALSE;
   IN_TRV_LIFT2.M_Adv_Err := FALSE;
   IN_TRV_LIFT2.M_Ret_Err := FALSE;
   IN_TRV_LIFT2.LP_Adv := FALSE;
   IN_TRV_LIFT2.LP_Ret := FALSE;
   IN_TRV_LIFT2.Visu_Adv := W#16#0;
   IN_TRV_LIFT2.Visu_Ret := W#16#0;
   IN_TRV_LIFT2.Error_T1.IN := FALSE;
   IN_TRV_LIFT2.Error_T1.PT := T#0MS;
   IN_TRV_LIFT2.Error_T1.Q := FALSE;
   IN_TRV_LIFT2.Error_T1.ET := T#0MS;
   IN_TRV_LIFT2.Error_T1.STATE := B#16#0;
   IN_TRV_LIFT2.Error_T1.STIME := T#0MS;
   IN_TRV_LIFT2.Error_T1.ATIME := T#0MS;
   IN_TRV_LIFT2.Error_T2.IN := FALSE;
   IN_TRV_LIFT2.Error_T2.PT := T#0MS;
   IN_TRV_LIFT2.Error_T2.Q := FALSE;
   IN_TRV_LIFT2.Error_T2.ET := T#0MS;
   IN_TRV_LIFT2.Error_T2.STATE := B#16#0;
   IN_TRV_LIFT2.Error_T2.STIME := T#0MS;
   IN_TRV_LIFT2.Error_T2.ATIME := T#0MS;
   IN_TRV_LIFT2.CHK_Aux1 := FALSE;
   IN_TRV_LIFT2.CHK_Aux2 := FALSE;
   IN_TRV_LIFT2.Error_T1_DN := FALSE;
   IN_TRV_LIFT2.Error_T2_DN := FALSE;
   IN_TRV_LIFT2.Adv_Memo := FALSE;
   IN_TRV_LIFT2.Visu_Adv_Arr[0] := FALSE;
   IN_TRV_LIFT2.Visu_Adv_Arr[1] := FALSE;
   IN_TRV_LIFT2.Visu_Adv_Arr[2] := FALSE;
   IN_TRV_LIFT2.Visu_Adv_Arr[3] := FALSE;
   IN_TRV_LIFT2.Visu_Adv_Arr[4] := FALSE;
   IN_TRV_LIFT2.Visu_Adv_Arr[5] := FALSE;
   IN_TRV_LIFT2.Visu_Adv_Arr[6] := FALSE;
   IN_TRV_LIFT2.Visu_Adv_Arr[7] := FALSE;
   IN_TRV_LIFT2.Visu_Adv_Arr[8] := FALSE;
   IN_TRV_LIFT2.Visu_Adv_Arr[9] := FALSE;
   IN_TRV_LIFT2.Visu_Adv_Arr[10] := FALSE;
   IN_TRV_LIFT2.Visu_Adv_Arr[11] := FALSE;
   IN_TRV_LIFT2.Visu_Adv_Arr[12] := FALSE;
   IN_TRV_LIFT2.Visu_Adv_Arr[13] := FALSE;
   IN_TRV_LIFT2.Visu_Adv_Arr[14] := FALSE;
   IN_TRV_LIFT2.Visu_Adv_Arr[15] := FALSE;
   IN_TRV_LIFT2.Visu_Ret_Arr[0] := FALSE;
   IN_TRV_LIFT2.Visu_Ret_Arr[1] := FALSE;
   IN_TRV_LIFT2.Visu_Ret_Arr[2] := FALSE;
   IN_TRV_LIFT2.Visu_Ret_Arr[3] := FALSE;
   IN_TRV_LIFT2.Visu_Ret_Arr[4] := FALSE;
   IN_TRV_LIFT2.Visu_Ret_Arr[5] := FALSE;
   IN_TRV_LIFT2.Visu_Ret_Arr[6] := FALSE;
   IN_TRV_LIFT2.Visu_Ret_Arr[7] := FALSE;
   IN_TRV_LIFT2.Visu_Ret_Arr[8] := FALSE;
   IN_TRV_LIFT2.Visu_Ret_Arr[9] := FALSE;
   IN_TRV_LIFT2.Visu_Ret_Arr[10] := FALSE;
   IN_TRV_LIFT2.Visu_Ret_Arr[11] := FALSE;
   IN_TRV_LIFT2.Visu_Ret_Arr[12] := FALSE;
   IN_TRV_LIFT2.Visu_Ret_Arr[13] := FALSE;
   IN_TRV_LIFT2.Visu_Ret_Arr[14] := FALSE;
   IN_TRV_LIFT2.Visu_Ret_Arr[15] := FALSE;
   IN_TRV_LIFT2.BLK_Move_Ret := 0;
   IN_TRV_LIFT2.Enable := FALSE;
   IN_TRV_LIFT2.Adv_End := FALSE;
   IN_TRV_LIFT2.Ret_End := FALSE;
   IN_TRV_ELE_AIR.Enable_Aux := FALSE;
   IN_TRV_ELE_AIR.Adv_Amount := 0;
   IN_TRV_ELE_AIR.Ret_Amount := 0;
   IN_TRV_ELE_AIR.LS_Adv1 := FALSE;
   IN_TRV_ELE_AIR.LS_Ret1 := FALSE;
   IN_TRV_ELE_AIR.LS_Adv2 := FALSE;
   IN_TRV_ELE_AIR.LS_Ret2 := FALSE;
   IN_TRV_ELE_AIR.LS_Adv3 := FALSE;
   IN_TRV_ELE_AIR.LS_Ret3 := FALSE;
   IN_TRV_ELE_AIR.LS_Adv4 := FALSE;
   IN_TRV_ELE_AIR.LS_Ret4 := FALSE;
   IN_TRV_ELE_AIR.SOL_Adv := FALSE;
   IN_TRV_ELE_AIR.SOL_Ret := FALSE;
   IN_TRV_ELE_AIR.M_Ready := FALSE;
   IN_TRV_ELE_AIR.T_CHK1 := T#0MS;
   IN_TRV_ELE_AIR.T_CHK2 := T#0MS;
   IN_TRV_ELE_AIR.PB_Lamp_CHK := FALSE;
   IN_TRV_ELE_AIR.PB_Error_Rst := FALSE;
   IN_TRV_ELE_AIR.M_FLICK := FALSE;
   IN_TRV_ELE_AIR.M_Adv_Err := FALSE;
   IN_TRV_ELE_AIR.M_Ret_Err := FALSE;
   IN_TRV_ELE_AIR.LP_Adv := FALSE;
   IN_TRV_ELE_AIR.LP_Ret := FALSE;
   IN_TRV_ELE_AIR.Visu_Adv := W#16#0;
   IN_TRV_ELE_AIR.Visu_Ret := W#16#0;
   IN_TRV_ELE_AIR.Error_T1.IN := FALSE;
   IN_TRV_ELE_AIR.Error_T1.PT := T#0MS;
   IN_TRV_ELE_AIR.Error_T1.Q := FALSE;
   IN_TRV_ELE_AIR.Error_T1.ET := T#0MS;
   IN_TRV_ELE_AIR.Error_T1.STATE := B#16#0;
   IN_TRV_ELE_AIR.Error_T1.STIME := T#0MS;
   IN_TRV_ELE_AIR.Error_T1.ATIME := T#0MS;
   IN_TRV_ELE_AIR.Error_T2.IN := FALSE;
   IN_TRV_ELE_AIR.Error_T2.PT := T#0MS;
   IN_TRV_ELE_AIR.Error_T2.Q := FALSE;
   IN_TRV_ELE_AIR.Error_T2.ET := T#0MS;
   IN_TRV_ELE_AIR.Error_T2.STATE := B#16#0;
   IN_TRV_ELE_AIR.Error_T2.STIME := T#0MS;
   IN_TRV_ELE_AIR.Error_T2.ATIME := T#0MS;
   IN_TRV_ELE_AIR.CHK_Aux1 := FALSE;
   IN_TRV_ELE_AIR.CHK_Aux2 := FALSE;
   IN_TRV_ELE_AIR.Error_T1_DN := FALSE;
   IN_TRV_ELE_AIR.Error_T2_DN := FALSE;
   IN_TRV_ELE_AIR.Adv_Memo := FALSE;
   IN_TRV_ELE_AIR.Visu_Adv_Arr[0] := FALSE;
   IN_TRV_ELE_AIR.Visu_Adv_Arr[1] := FALSE;
   IN_TRV_ELE_AIR.Visu_Adv_Arr[2] := FALSE;
   IN_TRV_ELE_AIR.Visu_Adv_Arr[3] := FALSE;
   IN_TRV_ELE_AIR.Visu_Adv_Arr[4] := FALSE;
   IN_TRV_ELE_AIR.Visu_Adv_Arr[5] := FALSE;
   IN_TRV_ELE_AIR.Visu_Adv_Arr[6] := FALSE;
   IN_TRV_ELE_AIR.Visu_Adv_Arr[7] := FALSE;
   IN_TRV_ELE_AIR.Visu_Adv_Arr[8] := FALSE;
   IN_TRV_ELE_AIR.Visu_Adv_Arr[9] := FALSE;
   IN_TRV_ELE_AIR.Visu_Adv_Arr[10] := FALSE;
   IN_TRV_ELE_AIR.Visu_Adv_Arr[11] := FALSE;
   IN_TRV_ELE_AIR.Visu_Adv_Arr[12] := FALSE;
   IN_TRV_ELE_AIR.Visu_Adv_Arr[13] := FALSE;
   IN_TRV_ELE_AIR.Visu_Adv_Arr[14] := FALSE;
   IN_TRV_ELE_AIR.Visu_Adv_Arr[15] := FALSE;
   IN_TRV_ELE_AIR.Visu_Ret_Arr[0] := FALSE;
   IN_TRV_ELE_AIR.Visu_Ret_Arr[1] := FALSE;
   IN_TRV_ELE_AIR.Visu_Ret_Arr[2] := FALSE;
   IN_TRV_ELE_AIR.Visu_Ret_Arr[3] := FALSE;
   IN_TRV_ELE_AIR.Visu_Ret_Arr[4] := FALSE;
   IN_TRV_ELE_AIR.Visu_Ret_Arr[5] := FALSE;
   IN_TRV_ELE_AIR.Visu_Ret_Arr[6] := FALSE;
   IN_TRV_ELE_AIR.Visu_Ret_Arr[7] := FALSE;
   IN_TRV_ELE_AIR.Visu_Ret_Arr[8] := FALSE;
   IN_TRV_ELE_AIR.Visu_Ret_Arr[9] := FALSE;
   IN_TRV_ELE_AIR.Visu_Ret_Arr[10] := FALSE;
   IN_TRV_ELE_AIR.Visu_Ret_Arr[11] := FALSE;
   IN_TRV_ELE_AIR.Visu_Ret_Arr[12] := FALSE;
   IN_TRV_ELE_AIR.Visu_Ret_Arr[13] := FALSE;
   IN_TRV_ELE_AIR.Visu_Ret_Arr[14] := FALSE;
   IN_TRV_ELE_AIR.Visu_Ret_Arr[15] := FALSE;
   IN_TRV_ELE_AIR.BLK_Move_Ret := 0;
   IN_TRV_ELE_AIR.Enable := FALSE;
   IN_TRV_ELE_AIR.Adv_End := FALSE;
   IN_TRV_ELE_AIR.Ret_End := FALSE;
END_DATA_BLOCK

FUNCTION FC 131 : VOID
TITLE =
VERSION : 0.1

BEGIN
NETWORK
TITLE =
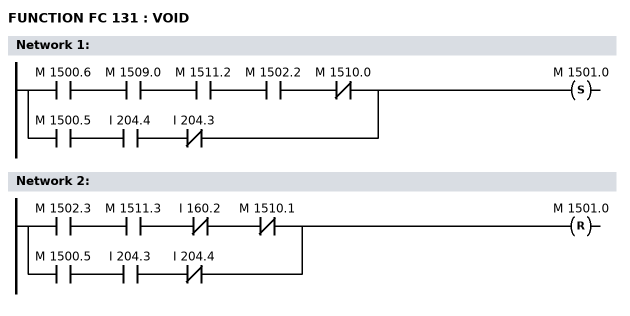

      A     M   1500.6;
      A     M   1509.0;
      A     M   1511.2;
      A     M   1502.2;
      AN    M   1510.0;
      O     ;
      A     M   1500.5;
      A     I    204.4;
      AN    I    204.3;
      S     M   1501.0;
NETWORK
TITLE =

      A     M   1502.3;
      A     M   1511.3;
      AN    I    160.2;
      AN    M   1510.1;
      O     ;
      A     M   1500.5;
      A     I    204.3;
      AN    I    204.4;
      R     M   1501.0;
END_FUNCTION

FUNCTION_BLOCK FB 132
TITLE =
VERSION : 0.1

BEGIN
NETWORK
TITLE =
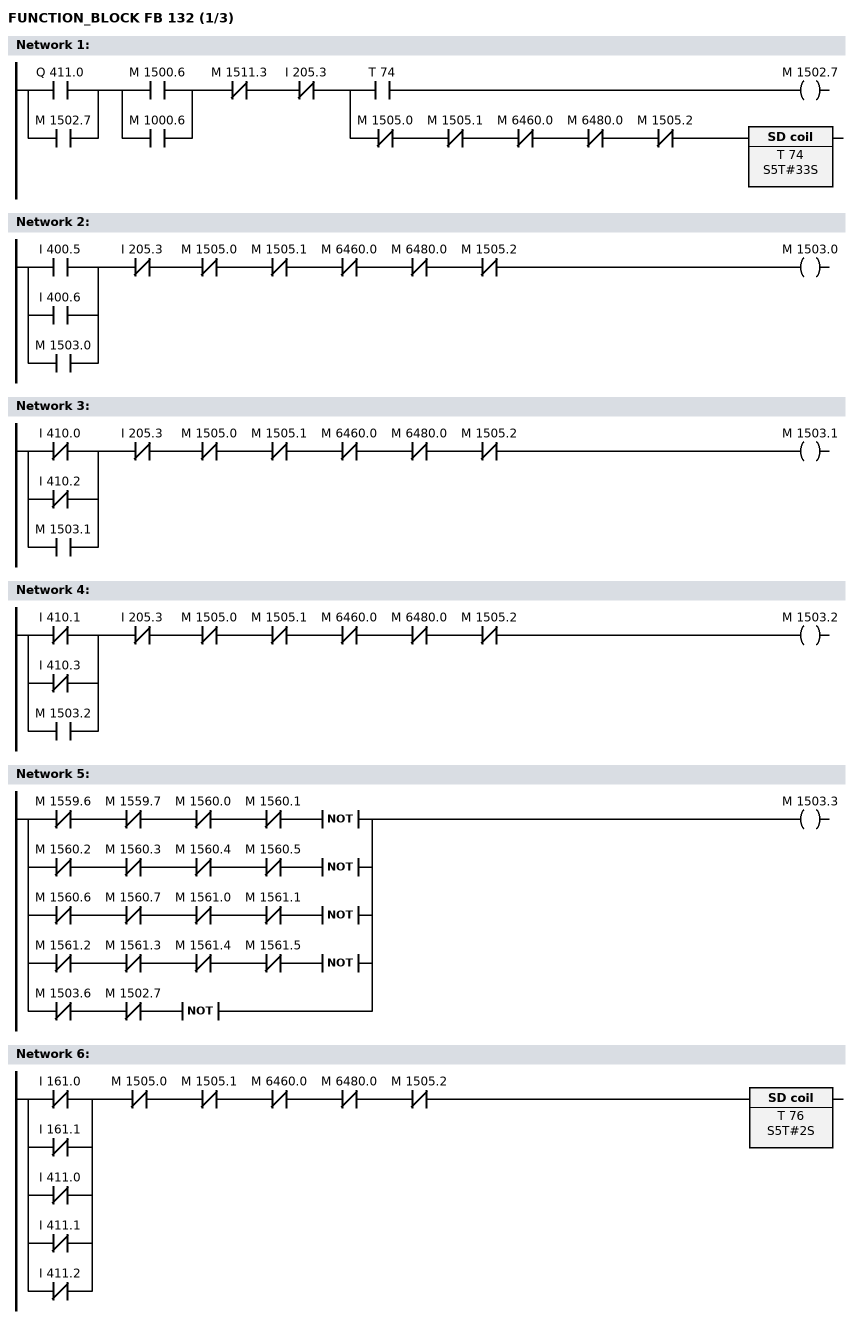

      A(    ;
      O     Q    411.0;
      O     M   1502.7;
      )     ;
      A(    ;
      O     M   1500.6;
      O     M   1000.6;
      )     ;
      AN    M   1511.3;
      AN    I    205.3;
      =     L      0.0;
      A     L      0.0;
      A     T     74;
      =     M   1502.7;
      A     L      0.0;
      AN    M   1505.0;
      AN    M   1505.1;
      AN    M   6460.0;
      AN    M   6480.0;
      AN    M   1505.2;
      L     S5T#33S;
      SD    T     74;
NETWORK
TITLE =

      A(    ;
      O     I    400.5;
      O     I    400.6;
      O     M   1503.0;
      )     ;
      AN    I    205.3;
      AN    M   1505.0;
      AN    M   1505.1;
      AN    M   6460.0;
      AN    M   6480.0;
      AN    M   1505.2;
      =     M   1503.0;
NETWORK
TITLE =

      A(    ;
      ON    I    410.0;
      ON    I    410.2;
      O     M   1503.1;
      )     ;
      AN    I    205.3;
      AN    M   1505.0;
      AN    M   1505.1;
      AN    M   6460.0;
      AN    M   6480.0;
      AN    M   1505.2;
      =     M   1503.1;
NETWORK
TITLE =

      A(    ;
      ON    I    410.1;
      ON    I    410.3;
      O     M   1503.2;
      )     ;
      AN    I    205.3;
      AN    M   1505.0;
      AN    M   1505.1;
      AN    M   6460.0;
      AN    M   6480.0;
      AN    M   1505.2;
      =     M   1503.2;
NETWORK
TITLE =

      AN    M   1559.6;
      AN    M   1559.7;
      AN    M   1560.0;
      AN    M   1560.1;
      NOT   ;
      O(    ;
      AN    M   1560.2;
      AN    M   1560.3;
      AN    M   1560.4;
      AN    M   1560.5;
      NOT   ;
      )     ;
      O(    ;
      AN    M   1560.6;
      AN    M   1560.7;
      AN    M   1561.0;
      AN    M   1561.1;
      NOT   ;
      )     ;
      O(    ;
      AN    M   1561.2;
      AN    M   1561.3;
      AN    M   1561.4;
      AN    M   1561.5;
      NOT   ;
      )     ;
      O(    ;
      AN    M   1503.6;
      AN    M   1502.7;
      NOT   ;
      )     ;
      =     M   1503.3;
NETWORK
TITLE =

      A(    ;
      ON    I    161.0;
      ON    I    161.1;
      ON    I    411.0;
      ON    I    411.1;
      ON    I    411.2;
      )     ;
      AN    M   1505.0;
      AN    M   1505.1;
      AN    M   6460.0;
      AN    M   6480.0;
      AN    M   1505.2;
      L     S5T#2S;
      SD    T     76;
NETWORK
TITLE =
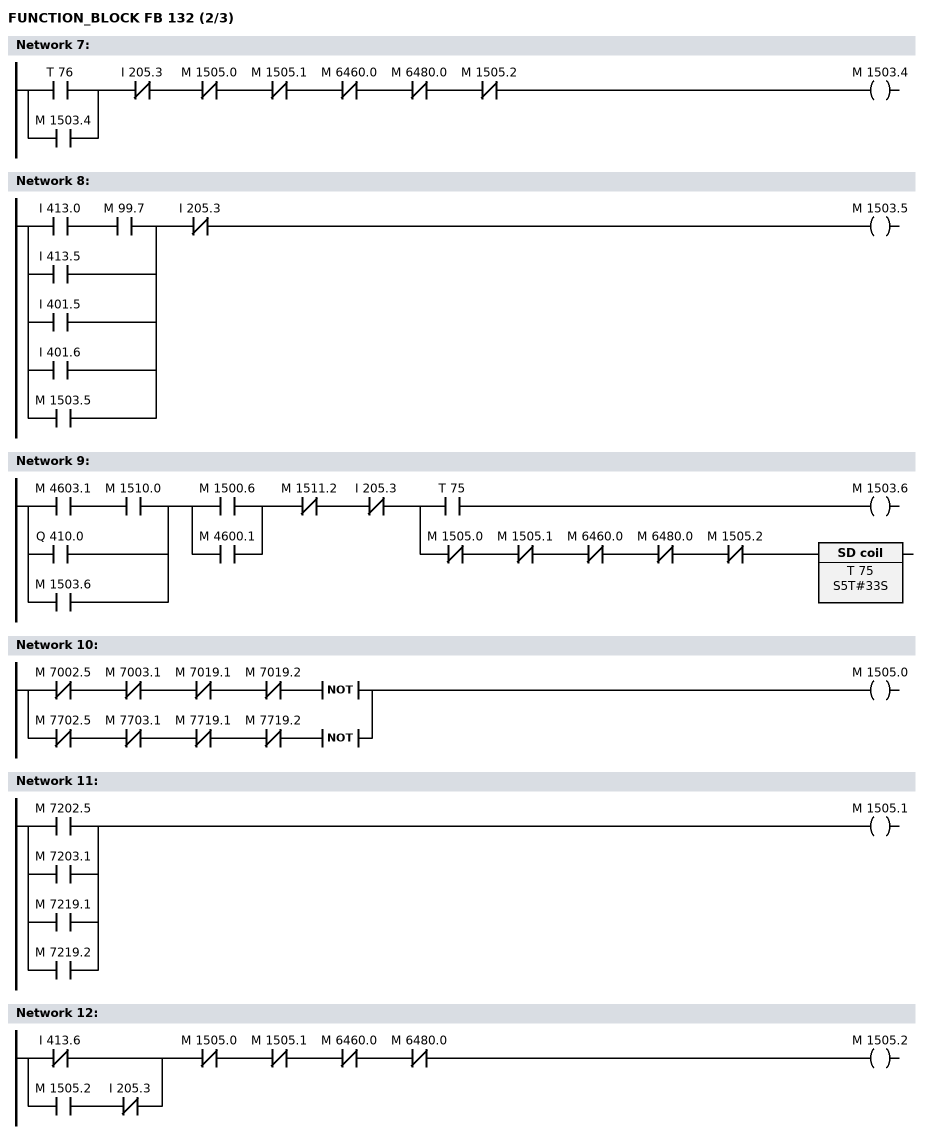

      A(    ;
      O     T     76;
      O     M   1503.4;
      )     ;
      AN    I    205.3;
      AN    M   1505.0;
      AN    M   1505.1;
      AN    M   6460.0;
      AN    M   6480.0;
      AN    M   1505.2;
      =     M   1503.4;
NETWORK
TITLE =

      A(    ;
      A     I    413.0;
      A     M     99.7;
      O     I    413.5;
      O     I    401.5;
      O     I    401.6;
      O     M   1503.5;
      )     ;
      AN    I    205.3;
      =     M   1503.5;
NETWORK
TITLE =

      A(    ;
      A     M   4603.1;
      A     M   1510.0;
      O     Q    410.0;
      O     M   1503.6;
      )     ;
      A(    ;
      O     M   1500.6;
      O     M   4600.1;
      )     ;
      AN    M   1511.2;
      AN    I    205.3;
      =     L      0.0;
      A     L      0.0;
      A     T     75;
      =     M   1503.6;
      A     L      0.0;
      AN    M   1505.0;
      AN    M   1505.1;
      AN    M   6460.0;
      AN    M   6480.0;
      AN    M   1505.2;
      L     S5T#33S;
      SD    T     75;
NETWORK
TITLE =

      AN    M   7002.5;
      AN    M   7003.1;
      AN    M   7019.1;
      AN    M   7019.2;
      NOT   ;
      O(    ;
      AN    M   7702.5;
      AN    M   7703.1;
      AN    M   7719.1;
      AN    M   7719.2;
      NOT   ;
      )     ;
      =     M   1505.0;
NETWORK
TITLE =

      O     M   7202.5;
      O     M   7203.1;
      O     M   7219.1;
      O     M   7219.2;
      =     M   1505.1;
NETWORK
TITLE =

      A(    ;
      ON    I    413.6;
      O     ;
      A     M   1505.2;
      AN    I    205.3;
      )     ;
      AN    M   1505.0;
      AN    M   1505.1;
      AN    M   6460.0;
      AN    M   6480.0;
      =     M   1505.2;
NETWORK
TITLE =
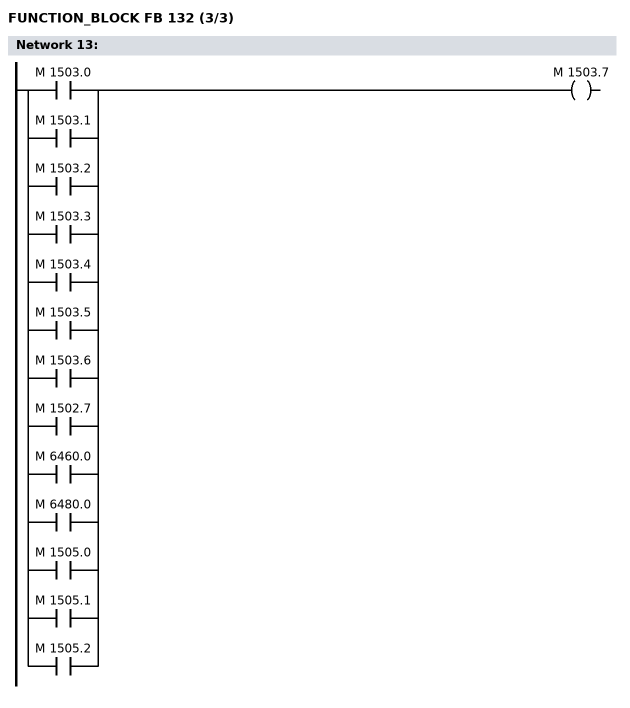

      O     M   1503.0;
      O     M   1503.1;
      O     M   1503.2;
      O     M   1503.3;
      O     M   1503.4;
      O     M   1503.5;
      O     M   1503.6;
      O     M   1502.7;
      O     M   6460.0;
      O     M   6480.0;
      O     M   1505.0;
      O     M   1505.1;
      O     M   1505.2;
      =     M   1503.7;
END_FUNCTION_BLOCK

DATA_BLOCK DB 132
TITLE =
VERSION : 0.0

 FB 132
BEGIN
END_DATA_BLOCK

FUNCTION FC 132 : VOID
TITLE =
VERSION : 0.1

BEGIN
NETWORK
TITLE =
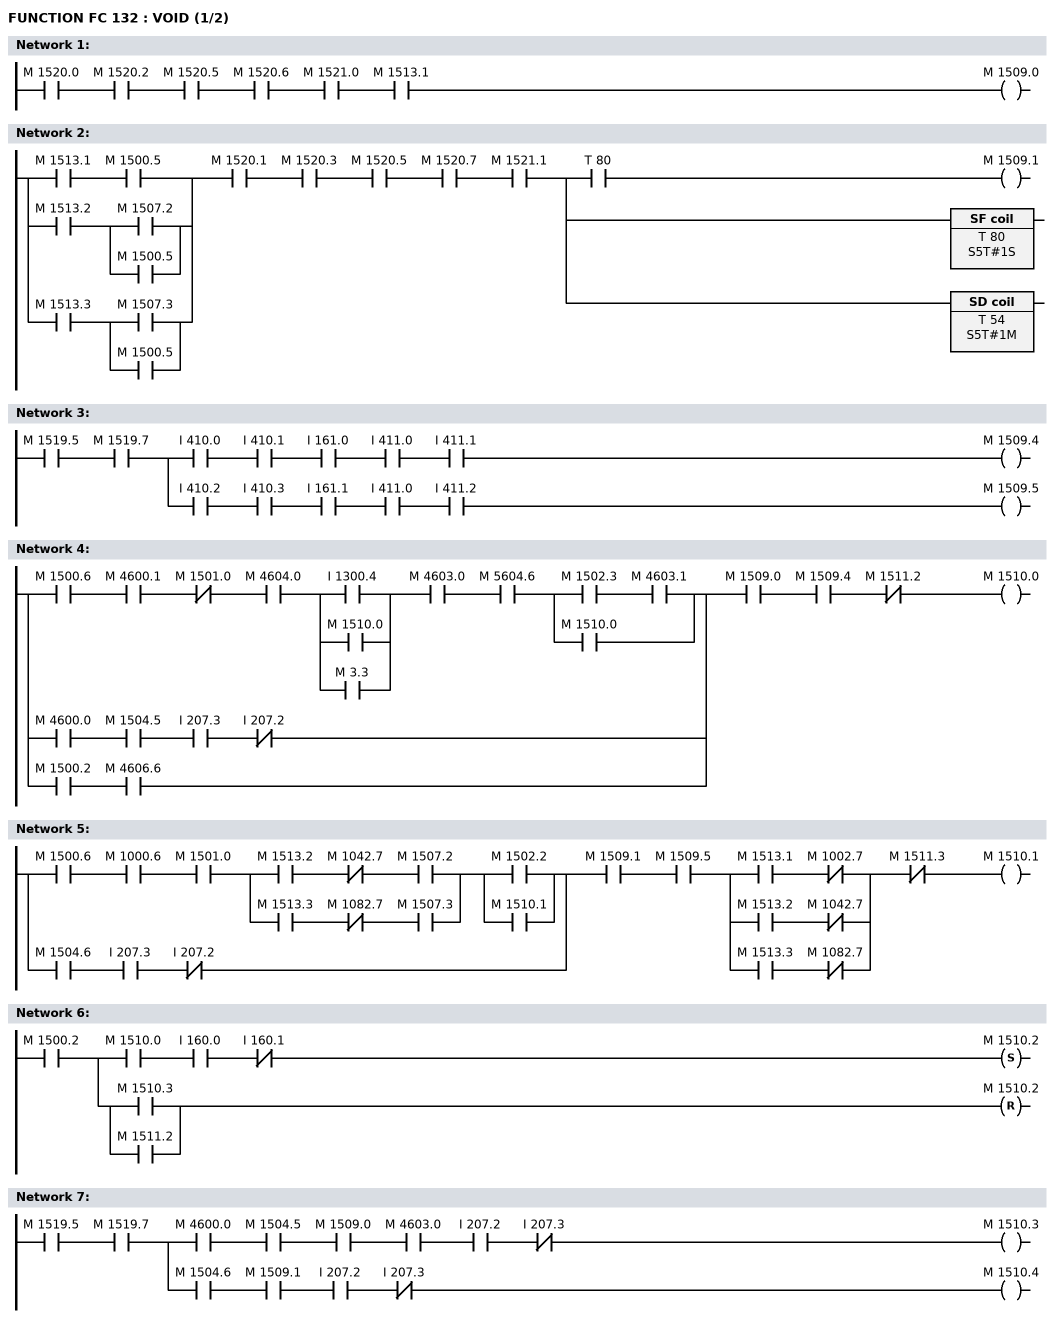

      A     M   1520.0;
      A     M   1520.2;
      A     M   1520.5;
      A     M   1520.6;
      A     M   1521.0;
      A     M   1513.1;
      =     M   1509.0;
NETWORK
TITLE =

      A(    ;
      A     M   1513.1;
      A     M   1500.5;
      O     ;
      A     M   1513.2;
      A(    ;
      O     M   1507.2;
      O     M   1500.5;
      )     ;
      O     ;
      A     M   1513.3;
      A(    ;
      O     M   1507.3;
      O     M   1500.5;
      )     ;
      )     ;
      A     M   1520.1;
      A     M   1520.3;
      A     M   1520.5;
      A     M   1520.7;
      A     M   1521.1;
      =     L      0.0;
      A     L      0.0;
      A     T     80;
      =     M   1509.1;
      A     L      0.0;
      BLD   102;
      L     S5T#1S;
      SF    T     80;
      A     L      0.0;
      BLD   102;
      L     S5T#1M;
      SD    T     54;
NETWORK
TITLE =

      A     M   1519.5;
      A     M   1519.7;
      =     L      0.0;
      A     L      0.0;
      A     I    410.0;
      A     I    410.1;
      A     I    161.0;
      A     I    411.0;
      A     I    411.1;
      =     M   1509.4;
      A     L      0.0;
      A     I    410.2;
      A     I    410.3;
      A     I    161.1;
      A     I    411.0;
      A     I    411.2;
      =     M   1509.5;
NETWORK
TITLE =

      A(    ;
      A     M   1500.6;
      A     M   4600.1;
      AN    M   1501.0;
      A     M   4604.0;
      A(    ;
      O     I   1300.4;
      O     M   1510.0;
      O     M      3.3;
      )     ;
      A     M   4603.0;
      A     M   5604.6;
      A(    ;
      A     M   1502.3;
      A     M   4603.1;
      O     M   1510.0;
      )     ;
      O     ;
      A     M   4600.0;
      A     M   1504.5;
      A     I    207.3;
      AN    I    207.2;
      O     ;
      A     M   1500.2;
      A     M   4606.6;
      )     ;
      A     M   1509.0;
      A     M   1509.4;
      AN    M   1511.2;
      =     M   1510.0;
NETWORK
TITLE =

      A(    ;
      A     M   1500.6;
      A     M   1000.6;
      A     M   1501.0;
      A(    ;
      A     M   1513.2;
      AN    M   1042.7;
      A     M   1507.2;
      O     ;
      A     M   1513.3;
      AN    M   1082.7;
      A     M   1507.3;
      )     ;
      A(    ;
      O     M   1502.2;
      O     M   1510.1;
      )     ;
      O     ;
      A     M   1504.6;
      A     I    207.3;
      AN    I    207.2;
      )     ;
      A     M   1509.1;
      A     M   1509.5;
      A(    ;
      A     M   1513.1;
      AN    M   1002.7;
      O     ;
      A     M   1513.2;
      AN    M   1042.7;
      O     ;
      A     M   1513.3;
      AN    M   1082.7;
      )     ;
      AN    M   1511.3;
      =     M   1510.1;
NETWORK
TITLE =

      A     M   1500.2;
      =     L      0.0;
      A     L      0.0;
      A     M   1510.0;
      A     I    160.0;
      AN    I    160.1;
      S     M   1510.2;
      A     L      0.0;
      A(    ;
      O     M   1510.3;
      O     M   1511.2;
      )     ;
      R     M   1510.2;
NETWORK
TITLE =

      A     M   1519.5;
      A     M   1519.7;
      =     L      0.0;
      A     L      0.0;
      A     M   4600.0;
      A     M   1504.5;
      A     M   1509.0;
      A     M   4603.0;
      A     I    207.2;
      AN    I    207.3;
      =     M   1510.3;
      A     L      0.0;
      A     M   1504.6;
      A     M   1509.1;
      A     I    207.2;
      AN    I    207.3;
      =     M   1510.4;
NETWORK
TITLE =
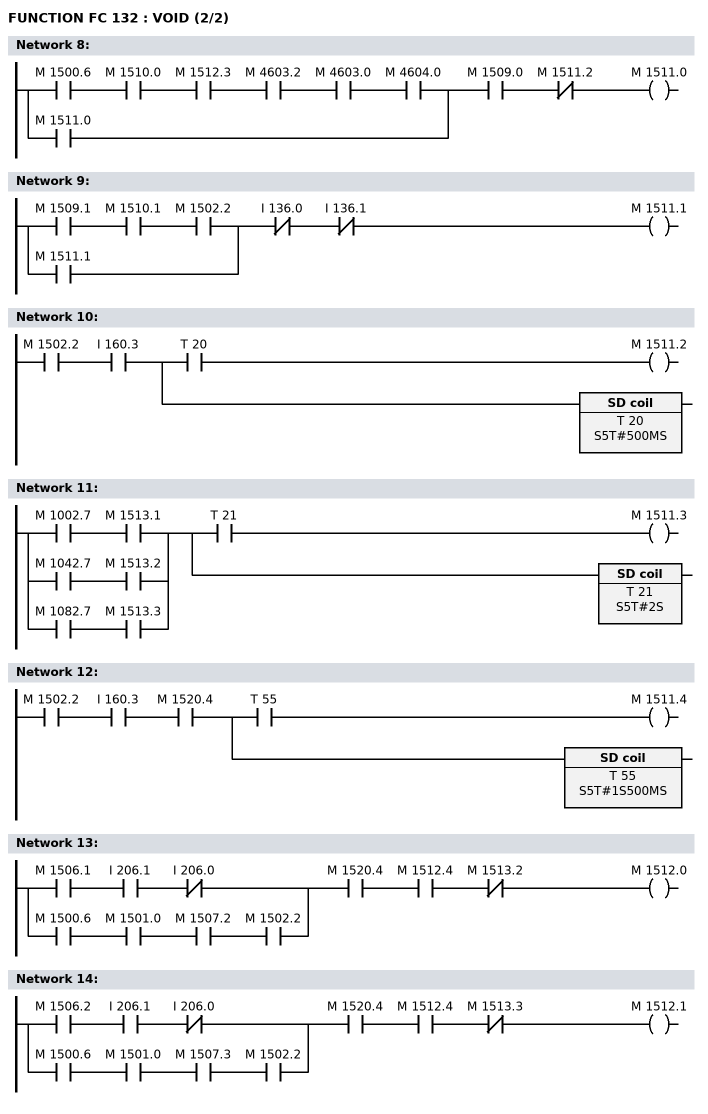

      A(    ;
      A     M   1500.6;
      A     M   1510.0;
      A     M   1512.3;
      A     M   4603.2;
      A     M   4603.0;
      A     M   4604.0;
      O     M   1511.0;
      )     ;
      A     M   1509.0;
      AN    M   1511.2;
      =     M   1511.0;
NETWORK
TITLE =

      A(    ;
      A     M   1509.1;
      A     M   1510.1;
      A     M   1502.2;
      O     M   1511.1;
      )     ;
      AN    I    136.0;
      AN    I    136.1;
      =     M   1511.1;
NETWORK
TITLE =

      A     M   1502.2;
      A     I    160.3;
      =     L      0.0;
      A     L      0.0;
      A     T     20;
      =     M   1511.2;
      A     L      0.0;
      BLD   102;
      L     S5T#500MS;
      SD    T     20;
NETWORK
TITLE =

      A     M   1002.7;
      A     M   1513.1;
      O     ;
      A     M   1042.7;
      A     M   1513.2;
      O     ;
      A     M   1082.7;
      A     M   1513.3;
      =     L      0.0;
      A     L      0.0;
      A     T     21;
      =     M   1511.3;
      A     L      0.0;
      BLD   102;
      L     S5T#2S;
      SD    T     21;
NETWORK
TITLE =

      A     M   1502.2;
      A     I    160.3;
      A     M   1520.4;
      =     L      0.0;
      A     L      0.0;
      A     T     55;
      =     M   1511.4;
      A     L      0.0;
      BLD   102;
      L     S5T#1S500MS;
      SD    T     55;
NETWORK
TITLE =

      A(    ;
      A     M   1506.1;
      A     I    206.1;
      AN    I    206.0;
      O     ;
      A     M   1500.6;
      A     M   1501.0;
      A     M   1507.2;
      A     M   1502.2;
      )     ;
      A     M   1520.4;
      A     M   1512.4;
      AN    M   1513.2;
      =     M   1512.0;
NETWORK
TITLE =

      A(    ;
      A     M   1506.2;
      A     I    206.1;
      AN    I    206.0;
      O     ;
      A     M   1500.6;
      A     M   1501.0;
      A     M   1507.3;
      A     M   1502.2;
      )     ;
      A     M   1520.4;
      A     M   1512.4;
      AN    M   1513.3;
      =     M   1512.1;
NETWORK
TITLE =

      A     M   1506.3;
      A     I    206.1;
      AN    I    206.0;
      A     M   1512.4;
      AN    M   1513.4;
      A     OV;
      =     M   1512.2;
NETWORK
TITLE =
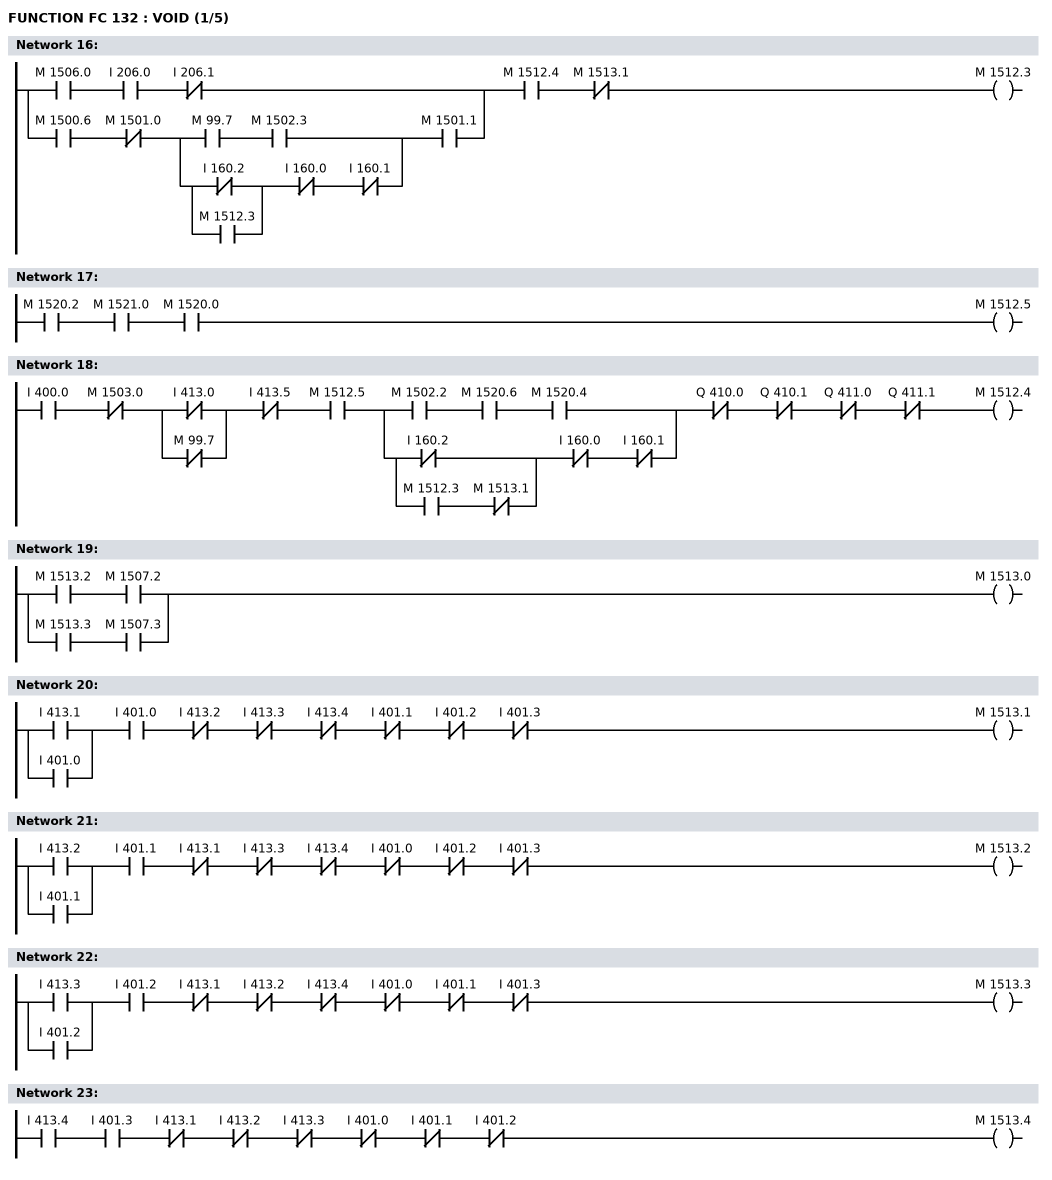

      A(    ;
      A     M   1506.0;
      A     I    206.0;
      AN    I    206.1;
      O     ;
      A     M   1500.6;
      AN    M   1501.0;
      A(    ;
      A     M     99.7;
      A     M   1502.3;
      O     ;
      A(    ;
      ON    I    160.2;
      O     M   1512.3;
      )     ;
      AN    I    160.0;
      AN    I    160.1;
      )     ;
      A     M   1501.1;
      )     ;
      A     M   1512.4;
      AN    M   1513.1;
      =     M   1512.3;
NETWORK
TITLE =

      A     M   1520.2;
      A     M   1521.0;
      A     M   1520.0;
      =     M   1512.5;
NETWORK
TITLE =

      A     I    400.0;
      AN    M   1503.0;
      A(    ;
      ON    I    413.0;
      ON    M     99.7;
      )     ;
      AN    I    413.5;
      A     M   1512.5;
      A(    ;
      A     M   1502.2;
      A     M   1520.6;
      A     M   1520.4;
      O     ;
      A(    ;
      ON    I    160.2;
      O     ;
      A     M   1512.3;
      AN    M   1513.1;
      )     ;
      AN    I    160.0;
      AN    I    160.1;
      )     ;
      AN    Q    410.0;
      AN    Q    410.1;
      AN    Q    411.0;
      AN    Q    411.1;
      =     M   1512.4;
NETWORK
TITLE =

      A     M   1513.2;
      A     M   1507.2;
      O     ;
      A     M   1513.3;
      A     M   1507.3;
      =     M   1513.0;
NETWORK
TITLE =

      A(    ;
      O     I    413.1;
      O     I    401.0;
      )     ;
      A     I    401.0;
      AN    I    413.2;
      AN    I    413.3;
      AN    I    413.4;
      AN    I    401.1;
      AN    I    401.2;
      AN    I    401.3;
      =     M   1513.1;
NETWORK
TITLE =

      A(    ;
      O     I    413.2;
      O     I    401.1;
      )     ;
      A     I    401.1;
      AN    I    413.1;
      AN    I    413.3;
      AN    I    413.4;
      AN    I    401.0;
      AN    I    401.2;
      AN    I    401.3;
      =     M   1513.2;
NETWORK
TITLE =

      A(    ;
      O     I    413.3;
      O     I    401.2;
      )     ;
      A     I    401.2;
      AN    I    413.1;
      AN    I    413.2;
      AN    I    413.4;
      AN    I    401.0;
      AN    I    401.1;
      AN    I    401.3;
      =     M   1513.3;
NETWORK
TITLE =

      A     I    413.4;
      A     I    401.3;
      AN    I    413.1;
      AN    I    413.2;
      AN    I    413.3;
      AN    I    401.0;
      AN    I    401.1;
      AN    I    401.2;
      =     M   1513.4;
NETWORK
TITLE =
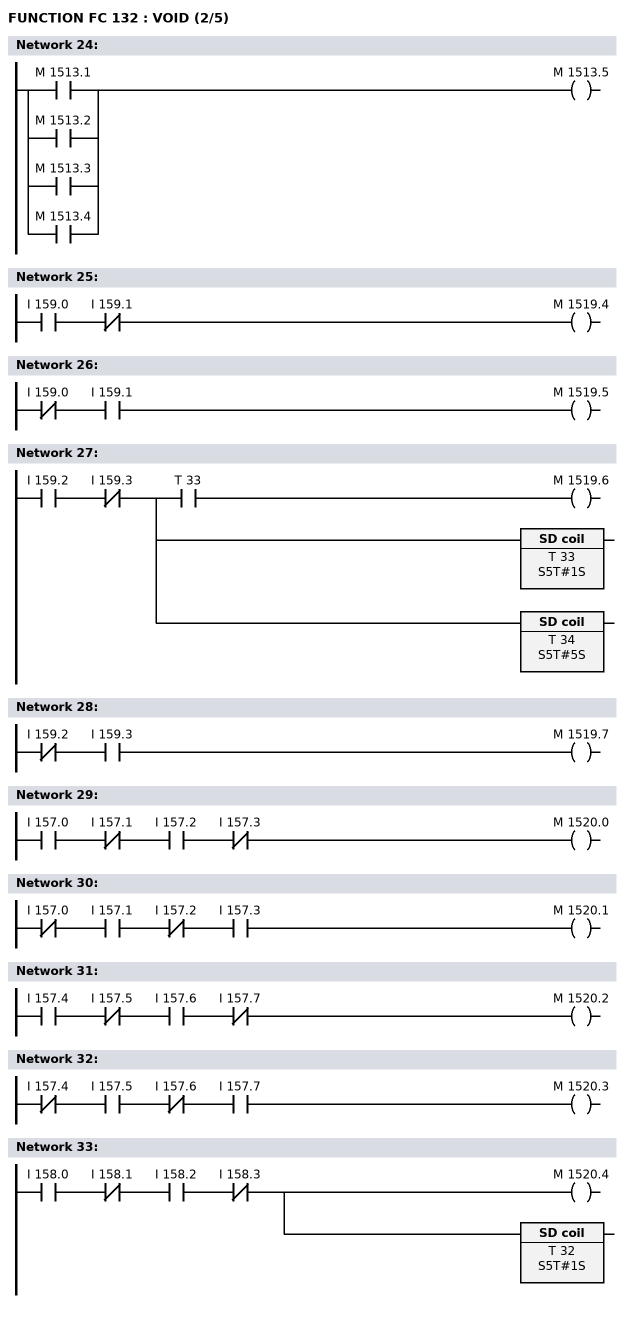

      O     M   1513.1;
      O     M   1513.2;
      O     M   1513.3;
      O     M   1513.4;
      =     M   1513.5;
NETWORK
TITLE =

      A     I    159.0;
      AN    I    159.1;
      =     M   1519.4;
NETWORK
TITLE =

      AN    I    159.0;
      A     I    159.1;
      =     M   1519.5;
NETWORK
TITLE =

      A     I    159.2;
      AN    I    159.3;
      =     L      0.0;
      A     L      0.0;
      A     T     33;
      =     M   1519.6;
      A     L      0.0;
      BLD   102;
      L     S5T#1S;
      SD    T     33;
      A     L      0.0;
      BLD   102;
      L     S5T#5S;
      SD    T     34;
NETWORK
TITLE =

      AN    I    159.2;
      A     I    159.3;
      =     M   1519.7;
NETWORK
TITLE =

      A     I    157.0;
      AN    I    157.1;
      A     I    157.2;
      AN    I    157.3;
      =     M   1520.0;
NETWORK
TITLE =

      AN    I    157.0;
      A     I    157.1;
      AN    I    157.2;
      A     I    157.3;
      =     M   1520.1;
NETWORK
TITLE =

      A     I    157.4;
      AN    I    157.5;
      A     I    157.6;
      AN    I    157.7;
      =     M   1520.2;
NETWORK
TITLE =

      AN    I    157.4;
      A     I    157.5;
      AN    I    157.6;
      A     I    157.7;
      =     M   1520.3;
NETWORK
TITLE =

      A     I    158.0;
      AN    I    158.1;
      A     I    158.2;
      AN    I    158.3;
      =     M   1520.4;
      L     S5T#1S;
      SD    T     32;
NETWORK
TITLE =
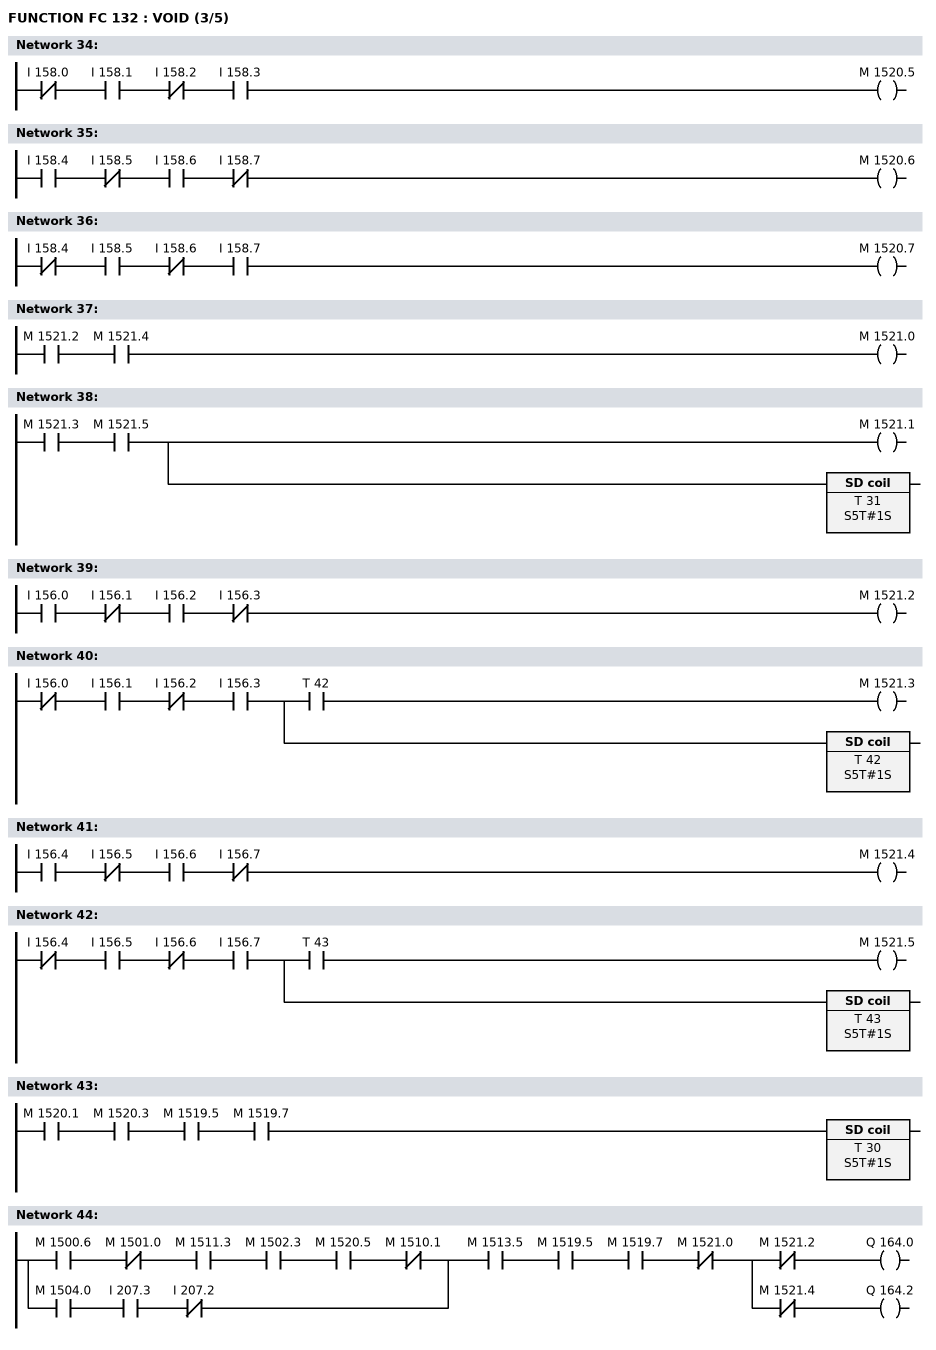

      AN    I    158.0;
      A     I    158.1;
      AN    I    158.2;
      A     I    158.3;
      =     M   1520.5;
NETWORK
TITLE =

      A     I    158.4;
      AN    I    158.5;
      A     I    158.6;
      AN    I    158.7;
      =     M   1520.6;
NETWORK
TITLE =

      AN    I    158.4;
      A     I    158.5;
      AN    I    158.6;
      A     I    158.7;
      =     M   1520.7;
NETWORK
TITLE =

      A     M   1521.2;
      A     M   1521.4;
      =     M   1521.0;
NETWORK
TITLE =

      A     M   1521.3;
      A     M   1521.5;
      =     M   1521.1;
      L     S5T#1S;
      SD    T     31;
NETWORK
TITLE =

      A     I    156.0;
      AN    I    156.1;
      A     I    156.2;
      AN    I    156.3;
      =     M   1521.2;
NETWORK
TITLE =

      AN    I    156.0;
      A     I    156.1;
      AN    I    156.2;
      A     I    156.3;
      =     L      0.0;
      A     L      0.0;
      A     T     42;
      =     M   1521.3;
      A     L      0.0;
      BLD   102;
      L     S5T#1S;
      SD    T     42;
NETWORK
TITLE =

      A     I    156.4;
      AN    I    156.5;
      A     I    156.6;
      AN    I    156.7;
      =     M   1521.4;
NETWORK
TITLE =

      AN    I    156.4;
      A     I    156.5;
      AN    I    156.6;
      A     I    156.7;
      =     L      0.0;
      A     L      0.0;
      A     T     43;
      =     M   1521.5;
      A     L      0.0;
      BLD   102;
      L     S5T#1S;
      SD    T     43;
NETWORK
TITLE =

      A     M   1520.1;
      A     M   1520.3;
      A     M   1519.5;
      A     M   1519.7;
      L     S5T#1S;
      SD    T     30;
NETWORK
TITLE =

      A(    ;
      A     M   1500.6;
      AN    M   1501.0;
      A     M   1511.3;
      A     M   1502.3;
      A     M   1520.5;
      AN    M   1510.1;
      O     ;
      A     M   1504.0;
      A     I    207.3;
      AN    I    207.2;
      )     ;
      A     M   1513.5;
      A     M   1519.5;
      A     M   1519.7;
      AN    M   1521.0;
      =     L      0.0;
      A     L      0.0;
      AN    M   1521.2;
      =     Q    164.0;
      A     L      0.0;
      AN    M   1521.4;
      =     Q    164.2;
NETWORK
TITLE =
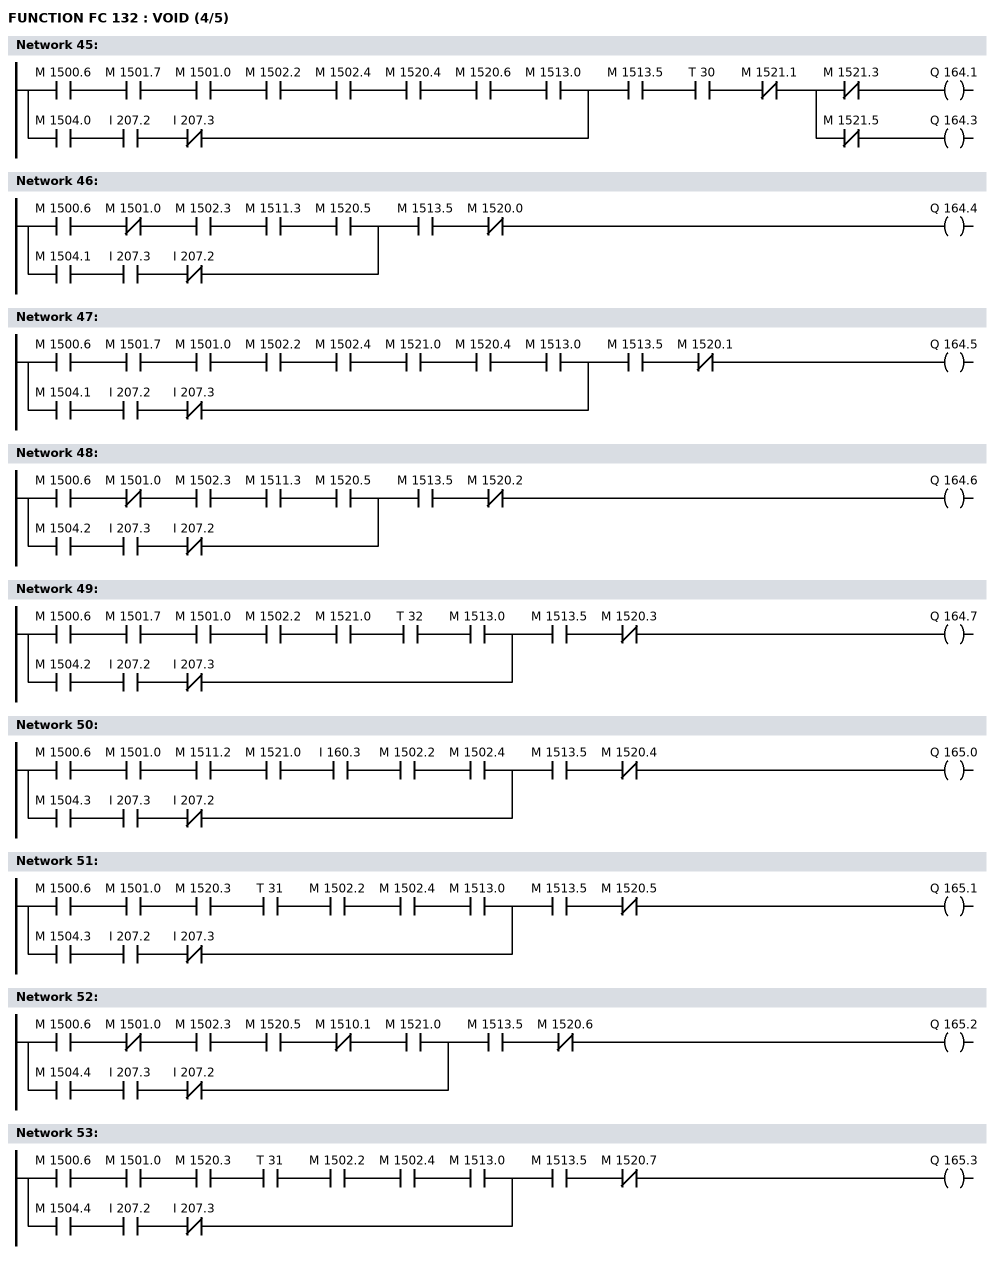

      A(    ;
      A     M   1500.6;
      A     M   1501.7;
      A     M   1501.0;
      A     M   1502.2;
      A     M   1502.4;
      A     M   1520.4;
      A     M   1520.6;
      A     M   1513.0;
      O     ;
      A     M   1504.0;
      A     I    207.2;
      AN    I    207.3;
      )     ;
      A     M   1513.5;
      A     T     30;
      AN    M   1521.1;
      =     L      0.0;
      A     L      0.0;
      AN    M   1521.3;
      =     Q    164.1;
      A     L      0.0;
      AN    M   1521.5;
      =     Q    164.3;
NETWORK
TITLE =

      A(    ;
      A     M   1500.6;
      AN    M   1501.0;
      A     M   1502.3;
      A     M   1511.3;
      A     M   1520.5;
      O     ;
      A     M   1504.1;
      A     I    207.3;
      AN    I    207.2;
      )     ;
      A     M   1513.5;
      AN    M   1520.0;
      =     Q    164.4;
NETWORK
TITLE =

      A(    ;
      A     M   1500.6;
      A     M   1501.7;
      A     M   1501.0;
      A     M   1502.2;
      A     M   1502.4;
      A     M   1521.0;
      A     M   1520.4;
      A     M   1513.0;
      O     ;
      A     M   1504.1;
      A     I    207.2;
      AN    I    207.3;
      )     ;
      A     M   1513.5;
      AN    M   1520.1;
      =     Q    164.5;
NETWORK
TITLE =

      A(    ;
      A     M   1500.6;
      AN    M   1501.0;
      A     M   1502.3;
      A     M   1511.3;
      A     M   1520.5;
      O     ;
      A     M   1504.2;
      A     I    207.3;
      AN    I    207.2;
      )     ;
      A     M   1513.5;
      AN    M   1520.2;
      =     Q    164.6;
NETWORK
TITLE =

      A(    ;
      A     M   1500.6;
      A     M   1501.7;
      A     M   1501.0;
      A     M   1502.2;
      A     M   1521.0;
      A     T     32;
      A     M   1513.0;
      O     ;
      A     M   1504.2;
      A     I    207.2;
      AN    I    207.3;
      )     ;
      A     M   1513.5;
      AN    M   1520.3;
      =     Q    164.7;
NETWORK
TITLE =

      A(    ;
      A     M   1500.6;
      A     M   1501.0;
      A     M   1511.2;
      A     M   1521.0;
      A     I    160.3;
      A     M   1502.2;
      A     M   1502.4;
      O     ;
      A     M   1504.3;
      A     I    207.3;
      AN    I    207.2;
      )     ;
      A     M   1513.5;
      AN    M   1520.4;
      =     Q    165.0;
NETWORK
TITLE =

      A(    ;
      A     M   1500.6;
      A     M   1501.0;
      A     M   1520.3;
      A     T     31;
      A     M   1502.2;
      A     M   1502.4;
      A     M   1513.0;
      O     ;
      A     M   1504.3;
      A     I    207.2;
      AN    I    207.3;
      )     ;
      A     M   1513.5;
      AN    M   1520.5;
      =     Q    165.1;
NETWORK
TITLE =

      A(    ;
      A     M   1500.6;
      AN    M   1501.0;
      A     M   1502.3;
      A     M   1520.5;
      AN    M   1510.1;
      A     M   1521.0;
      O     ;
      A     M   1504.4;
      A     I    207.3;
      AN    I    207.2;
      )     ;
      A     M   1513.5;
      AN    M   1520.6;
      =     Q    165.2;
NETWORK
TITLE =

      A(    ;
      A     M   1500.6;
      A     M   1501.0;
      A     M   1520.3;
      A     T     31;
      A     M   1502.2;
      A     M   1502.4;
      A     M   1513.0;
      O     ;
      A     M   1504.4;
      A     I    207.2;
      AN    I    207.3;
      )     ;
      A     M   1513.5;
      AN    M   1520.7;
      =     Q    165.3;
NETWORK
TITLE =
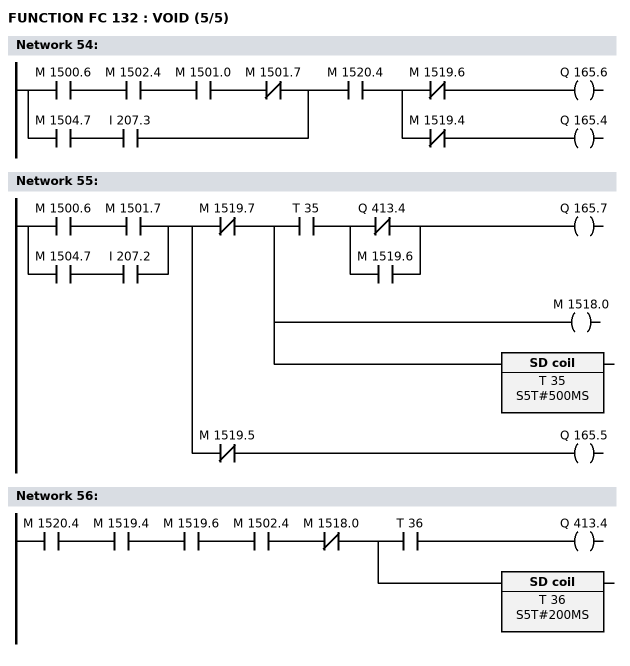

      A(    ;
      A     M   1500.6;
      A     M   1502.4;
      A     M   1501.0;
      AN    M   1501.7;
      O     ;
      A     M   1504.7;
      A     I    207.3;
      )     ;
      A     M   1520.4;
      =     L      0.0;
      A     L      0.0;
      AN    M   1519.6;
      =     Q    165.6;
      A     L      0.0;
      AN    M   1519.4;
      =     Q    165.4;
NETWORK
TITLE =

      A     M   1500.6;
      A     M   1501.7;
      O     ;
      A     M   1504.7;
      A     I    207.2;
      =     L      0.0;
      A     L      0.0;
      AN    M   1519.7;
      =     L      0.1;
      A     L      0.1;
      A     T     35;
      A(    ;
      ON    Q    413.4;
      O     M   1519.6;
      )     ;
      =     Q    165.7;
      A     L      0.1;
      BLD   102;
      =     M   1518.0;
      A     L      0.1;
      BLD   102;
      L     S5T#500MS;
      SD    T     35;
      A     L      0.0;
      AN    M   1519.5;
      =     Q    165.5;
NETWORK
TITLE =

      A     M   1520.4;
      A     M   1519.4;
      A     M   1519.6;
      A     M   1502.4;
      AN    M   1518.0;
      =     L      0.0;
      A     L      0.0;
      A     T     36;
      =     Q    413.4;
      A     L      0.0;
      BLD   102;
      L     S5T#200MS;
      SD    T     36;
END_FUNCTION

FUNCTION FC 133 : VOID
TITLE =
VERSION : 0.1

BEGIN
NETWORK
TITLE =

      AN    I    401.7;
      A(    ;
      O     M   1512.0;
      O     M   1512.1;
      O     ;
      A     M   1512.2;
      A     OV;
      O     M   1512.3;
      )     ;
      =     Q    400.0;
NETWORK
TITLE =
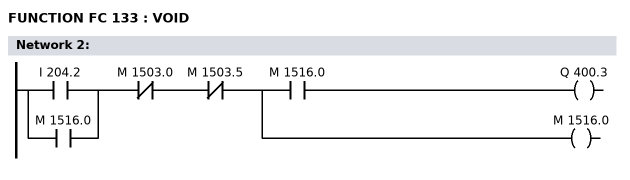

      A(    ;
      O     I    204.2;
      O     M   1516.0;
      )     ;
      AN    M   1503.0;
      AN    M   1503.5;
      =     L      0.0;
      A     L      0.0;
      A     M   1516.0;
      =     Q    400.3;
      A     L      0.0;
      BLD   102;
      =     M   1516.0;
NETWORK
TITLE =

      AN    I    401.7;
      A(    ;
      O     M   1512.0;
      O     M   1512.1;
      O     ;
      A     M   1512.2;
      A     OV;
      O     M   1512.3;
      )     ;
      =     L      0.0;
      A     L      0.0;
      A     T     41;
      AN    T     40;
      =     Q    400.4;
      A     L      0.0;
      BLD   102;
      L     S5T#2S;
      SD    T     40;
      A     L      0.0;
      BLD   102;
      L     S5T#500MS;
      SD    T     41;
NETWORK
TITLE =

      AN    M   1500.0;
      =     Q    401.5;
NETWORK
TITLE =

      A     M   1516.0;
      AN    I    401.7;
      =     L      0.0;
      A     L      0.0;
      A(    ;
      O     M   1506.0;
      O     M   1512.3;
      )     ;
      =     Q    402.0;
      A     L      0.0;
      A(    ;
      O     M   1506.1;
      O     M   1512.0;
      )     ;
      =     Q    402.1;
      A     L      0.0;
      A(    ;
      O     M   1506.2;
      O     M   1512.1;
      )     ;
      =     Q    402.2;
      A     L      0.0;
      A     M   1506.3;
      A     OV;
      =     Q    402.3;
NETWORK
TITLE =
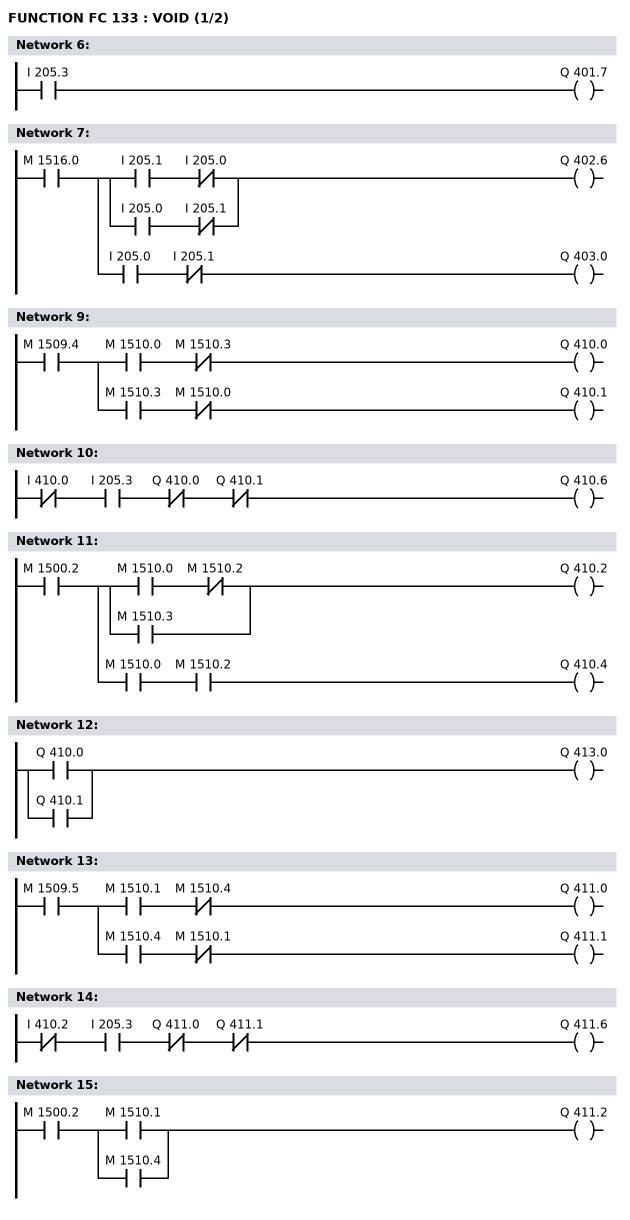

      A     I    205.3;
      =     Q    401.7;
NETWORK
TITLE =

      A     M   1516.0;
      =     L      0.0;
      A     L      0.0;
      A(    ;
      A     I    205.1;
      AN    I    205.0;
      O     ;
      A     I    205.0;
      AN    I    205.1;
      )     ;
      =     Q    402.6;
      A     L      0.0;
      A     I    205.0;
      AN    I    205.1;
      =     Q    403.0;
NETWORK
TITLE =

NETWORK
TITLE =

      A     M   1509.4;
      =     L      0.0;
      A     L      0.0;
      A     M   1510.0;
      AN    M   1510.3;
      =     Q    410.0;
      A     L      0.0;
      A     M   1510.3;
      AN    M   1510.0;
      =     Q    410.1;
NETWORK
TITLE =

      AN    I    410.0;
      A     I    205.3;
      AN    Q    410.0;
      AN    Q    410.1;
      =     Q    410.6;
NETWORK
TITLE =

      A     M   1500.2;
      =     L      0.0;
      A     L      0.0;
      A(    ;
      A     M   1510.0;
      AN    M   1510.2;
      O     M   1510.3;
      )     ;
      =     Q    410.2;
      A     L      0.0;
      A     M   1510.0;
      A     M   1510.2;
      =     Q    410.4;
NETWORK
TITLE =

      O     Q    410.0;
      O     Q    410.1;
      =     Q    413.0;
NETWORK
TITLE =

      A     M   1509.5;
      =     L      0.0;
      A     L      0.0;
      A     M   1510.1;
      AN    M   1510.4;
      =     Q    411.0;
      A     L      0.0;
      A     M   1510.4;
      AN    M   1510.1;
      =     Q    411.1;
NETWORK
TITLE =

      AN    I    410.2;
      A     I    205.3;
      AN    Q    411.0;
      AN    Q    411.1;
      =     Q    411.6;
NETWORK
TITLE =

      A     M   1500.2;
      A(    ;
      O     M   1510.1;
      O     M   1510.4;
      )     ;
      =     Q    411.2;
NETWORK
TITLE =
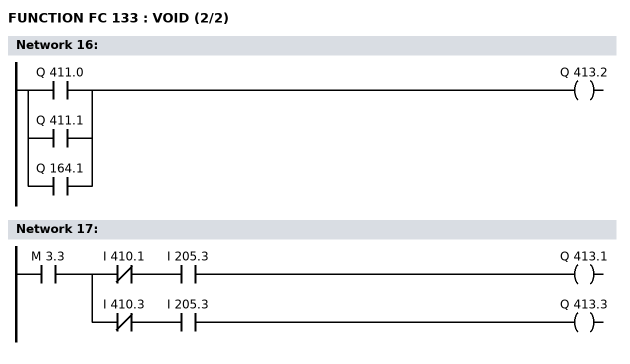

      O     Q    411.0;
      O     Q    411.1;
      O     Q    164.1;
      =     Q    413.2;
NETWORK
TITLE =

      A     M      3.3;
      =     L      0.0;
      A     L      0.0;
      AN    I    410.1;
      A     I    205.3;
      =     Q    413.1;
      A     L      0.0;
      AN    I    410.3;
      A     I    205.3;
      =     Q    413.3;
END_FUNCTION

FUNCTION_BLOCK FB 140
TITLE =
VERSION : 0.1

BEGIN
NETWORK
TITLE =

END_FUNCTION_BLOCK

FUNCTION FC 140 : VOID
TITLE =
VERSION : 0.1

BEGIN
NETWORK
TITLE =

END_FUNCTION

FUNCTION_BLOCK FB 141
TITLE =
VERSION : 0.1

BEGIN
NETWORK
TITLE =

END_FUNCTION_BLOCK

FUNCTION FC 141 : VOID
TITLE =
VERSION : 0.1

BEGIN
NETWORK
TITLE =

END_FUNCTION

FUNCTION_BLOCK FB 142
TITLE =
VERSION : 0.1

BEGIN
NETWORK
TITLE =

END_FUNCTION_BLOCK

FUNCTION FC 142 : VOID
TITLE =
VERSION : 0.1

BEGIN
NETWORK
TITLE =

END_FUNCTION

FUNCTION FC 146 : VOID
TITLE =
VERSION : 0.1

BEGIN
NETWORK
TITLE =
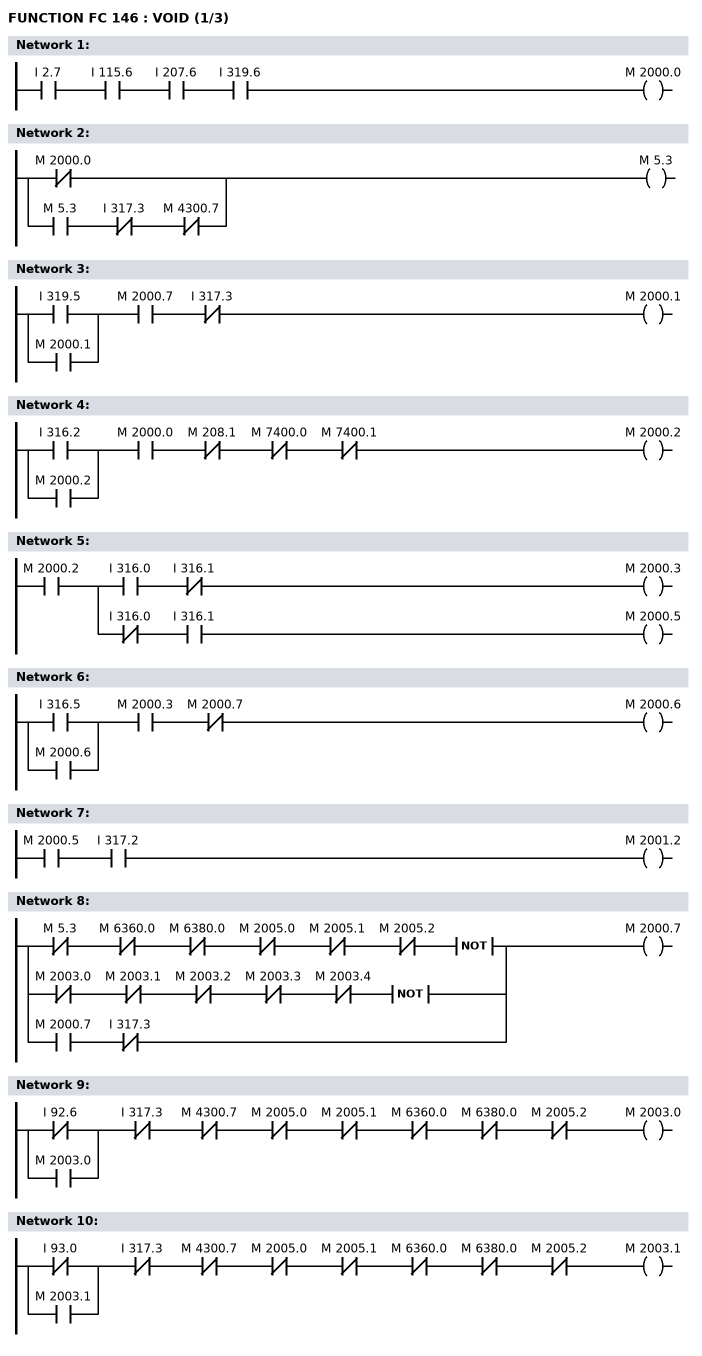

      A     I      2.7;
      A     I    115.6;
      A     I    207.6;
      A     I    319.6;
      =     M   2000.0;
NETWORK
TITLE =

      ON    M   2000.0;
      O     ;
      A     M      5.3;
      AN    I    317.3;
      AN    M   4300.7;
      =     M      5.3;
NETWORK
TITLE =

      A(    ;
      O     I    319.5;
      O     M   2000.1;
      )     ;
      A     M   2000.7;
      AN    I    317.3;
      =     M   2000.1;
NETWORK
TITLE =

      A(    ;
      O     I    316.2;
      O     M   2000.2;
      )     ;
      A     M   2000.0;
      AN    M    208.1;
      AN    M   7400.0;
      AN    M   7400.1;
      =     M   2000.2;
NETWORK
TITLE =

      A     M   2000.2;
      =     L      0.0;
      A     L      0.0;
      A     I    316.0;
      AN    I    316.1;
      =     M   2000.3;
      A     L      0.0;
      AN    I    316.0;
      A     I    316.1;
      =     M   2000.5;
NETWORK
TITLE =

      A(    ;
      O     I    316.5;
      O     M   2000.6;
      )     ;
      A     M   2000.3;
      AN    M   2000.7;
      =     M   2000.6;
NETWORK
TITLE =

      A     M   2000.5;
      A     I    317.2;
      =     M   2001.2;
NETWORK
TITLE =

      AN    M      5.3;
      AN    M   6360.0;
      AN    M   6380.0;
      AN    M   2005.0;
      AN    M   2005.1;
      AN    M   2005.2;
      NOT   ;
      O(    ;
      AN    M   2003.0;
      AN    M   2003.1;
      AN    M   2003.2;
      AN    M   2003.3;
      AN    M   2003.4;
      NOT   ;
      )     ;
      O     ;
      A     M   2000.7;
      AN    I    317.3;
      =     M   2000.7;
NETWORK
TITLE =

      A(    ;
      ON    I     92.6;
      O     M   2003.0;
      )     ;
      AN    I    317.3;
      AN    M   4300.7;
      AN    M   2005.0;
      AN    M   2005.1;
      AN    M   6360.0;
      AN    M   6380.0;
      AN    M   2005.2;
      =     M   2003.0;
NETWORK
TITLE =

      A(    ;
      ON    I     93.0;
      O     M   2003.1;
      )     ;
      AN    I    317.3;
      AN    M   4300.7;
      AN    M   2005.0;
      AN    M   2005.1;
      AN    M   6360.0;
      AN    M   6380.0;
      AN    M   2005.2;
      =     M   2003.1;
NETWORK
TITLE =
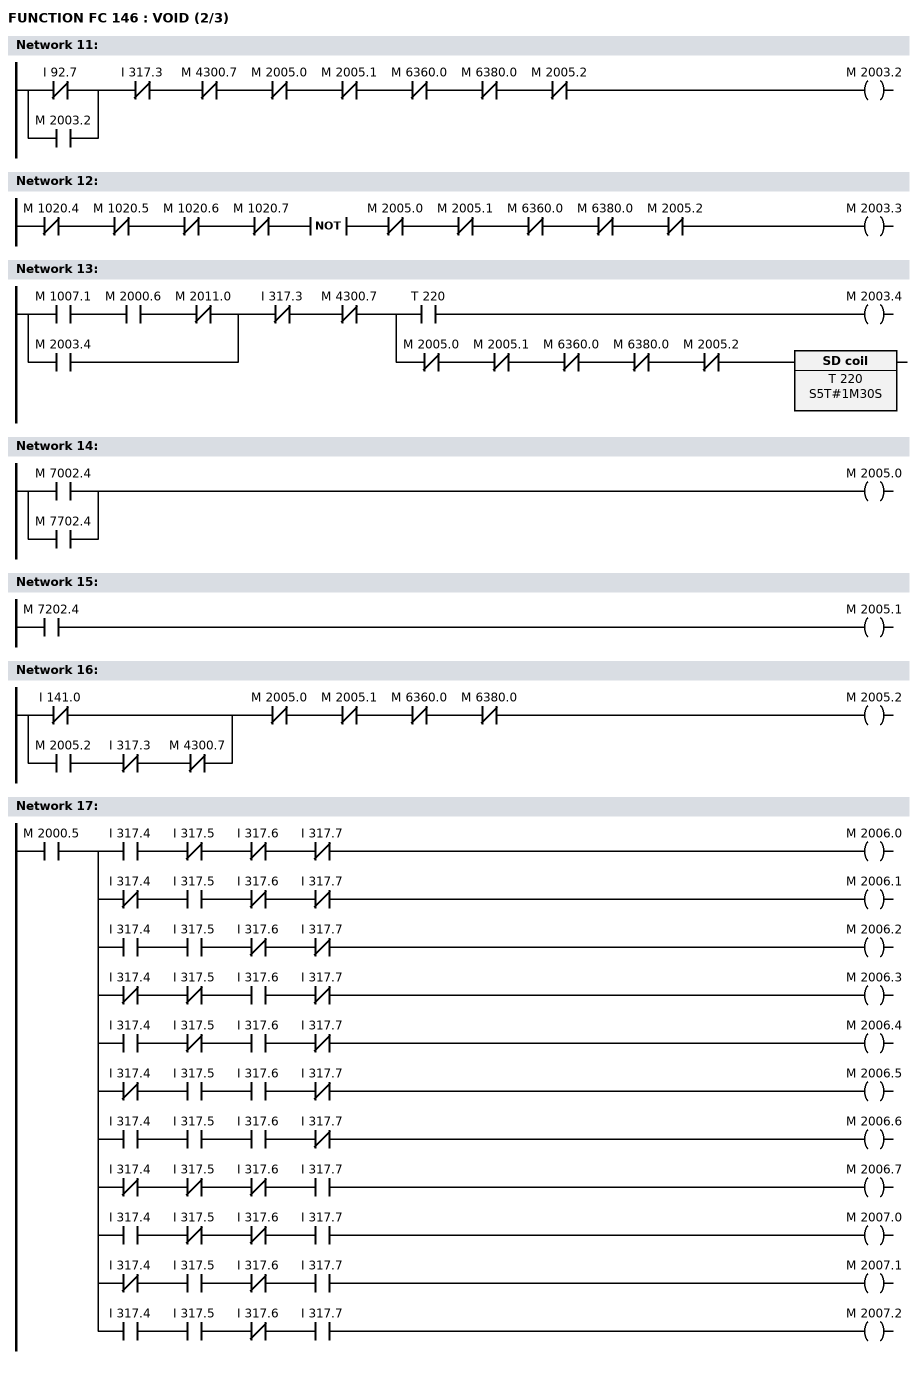

      A(    ;
      ON    I     92.7;
      O     M   2003.2;
      )     ;
      AN    I    317.3;
      AN    M   4300.7;
      AN    M   2005.0;
      AN    M   2005.1;
      AN    M   6360.0;
      AN    M   6380.0;
      AN    M   2005.2;
      =     M   2003.2;
NETWORK
TITLE =

      AN    M   1020.4;
      AN    M   1020.5;
      AN    M   1020.6;
      AN    M   1020.7;
      NOT   ;
      AN    M   2005.0;
      AN    M   2005.1;
      AN    M   6360.0;
      AN    M   6380.0;
      AN    M   2005.2;
      =     M   2003.3;
NETWORK
TITLE =

      A(    ;
      A     M   1007.1;
      A     M   2000.6;
      AN    M   2011.0;
      O     M   2003.4;
      )     ;
      AN    I    317.3;
      AN    M   4300.7;
      =     L      0.0;
      A     L      0.0;
      A     T    220;
      =     M   2003.4;
      A     L      0.0;
      AN    M   2005.0;
      AN    M   2005.1;
      AN    M   6360.0;
      AN    M   6380.0;
      AN    M   2005.2;
      L     S5T#1M30S;
      SD    T    220;
NETWORK
TITLE =

      O     M   7002.4;
      O     M   7702.4;
      =     M   2005.0;
NETWORK
TITLE =

      A     M   7202.4;
      =     M   2005.1;
NETWORK
TITLE =

      A(    ;
      ON    I    141.0;
      O     ;
      A     M   2005.2;
      AN    I    317.3;
      AN    M   4300.7;
      )     ;
      AN    M   2005.0;
      AN    M   2005.1;
      AN    M   6360.0;
      AN    M   6380.0;
      =     M   2005.2;
NETWORK
TITLE =

      A     M   2000.5;
      =     L      0.0;
      A     L      0.0;
      A     I    317.4;
      AN    I    317.5;
      AN    I    317.6;
      AN    I    317.7;
      =     M   2006.0;
      A     L      0.0;
      AN    I    317.4;
      A     I    317.5;
      AN    I    317.6;
      AN    I    317.7;
      =     M   2006.1;
      A     L      0.0;
      A     I    317.4;
      A     I    317.5;
      AN    I    317.6;
      AN    I    317.7;
      =     M   2006.2;
      A     L      0.0;
      AN    I    317.4;
      AN    I    317.5;
      A     I    317.6;
      AN    I    317.7;
      =     M   2006.3;
      A     L      0.0;
      A     I    317.4;
      AN    I    317.5;
      A     I    317.6;
      AN    I    317.7;
      =     M   2006.4;
      A     L      0.0;
      AN    I    317.4;
      A     I    317.5;
      A     I    317.6;
      AN    I    317.7;
      =     M   2006.5;
      A     L      0.0;
      A     I    317.4;
      A     I    317.5;
      A     I    317.6;
      AN    I    317.7;
      =     M   2006.6;
      A     L      0.0;
      AN    I    317.4;
      AN    I    317.5;
      AN    I    317.6;
      A     I    317.7;
      =     M   2006.7;
      A     L      0.0;
      A     I    317.4;
      AN    I    317.5;
      AN    I    317.6;
      A     I    317.7;
      =     M   2007.0;
      A     L      0.0;
      AN    I    317.4;
      A     I    317.5;
      AN    I    317.6;
      A     I    317.7;
      =     M   2007.1;
      A     L      0.0;
      A     I    317.4;
      A     I    317.5;
      AN    I    317.6;
      A     I    317.7;
      =     M   2007.2;
NETWORK
TITLE =
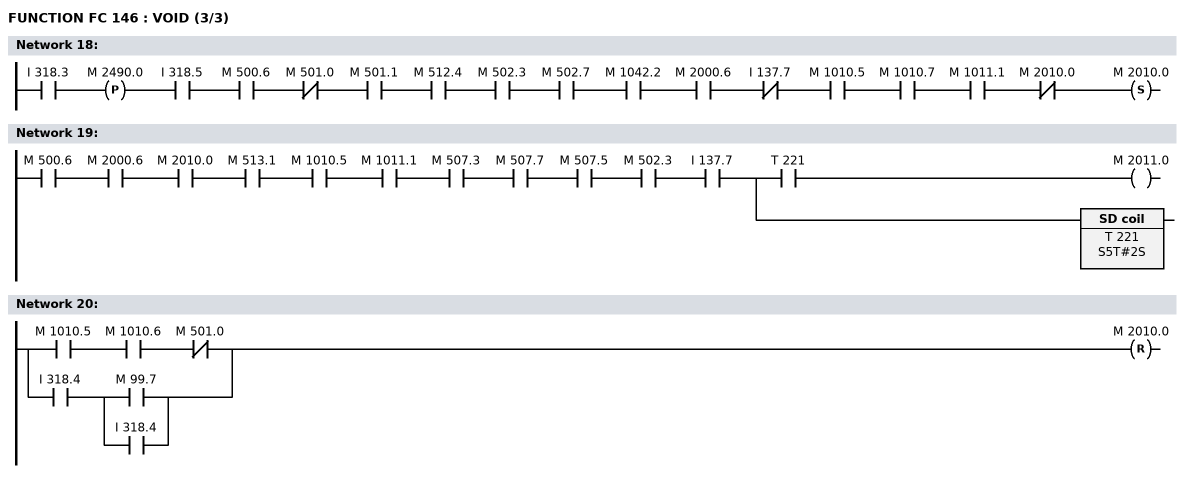

      A     I    318.3;
      FP    M   2490.0;
      A     I    318.5;
      A     M    500.6;
      AN    M    501.0;
      A     M    501.1;
      A     M    512.4;
      A     M    502.3;
      A     M    502.7;
      A     M   1042.2;
      A     M   2000.6;
      AN    I    137.7;
      A     M   1010.5;
      A     M   1010.7;
      A     M   1011.1;
      AN    M   2010.0;
      S     M   2010.0;
NETWORK
TITLE =

      A     M    500.6;
      A     M   2000.6;
      A     M   2010.0;
      A     M    513.1;
      A     M   1010.5;
      A     M   1011.1;
      A     M    507.3;
      A     M    507.7;
      A     M    507.5;
      A     M    502.3;
      A     I    137.7;
      =     L      0.0;
      A     L      0.0;
      A     T    221;
      =     M   2011.0;
      A     L      0.0;
      BLD   102;
      L     S5T#2S;
      SD    T    221;
NETWORK
TITLE =

      A     M   1010.5;
      A     M   1010.6;
      AN    M    501.0;
      O     ;
      A     I    318.4;
      A(    ;
      O     M     99.7;
      O     I    318.4;
      )     ;
      R     M   2010.0;
END_FUNCTION

FUNCTION FC 160 : VOID
TITLE =
VERSION : 0.1

BEGIN
NETWORK
TITLE =리턴라인 표준 조작반 LAMP
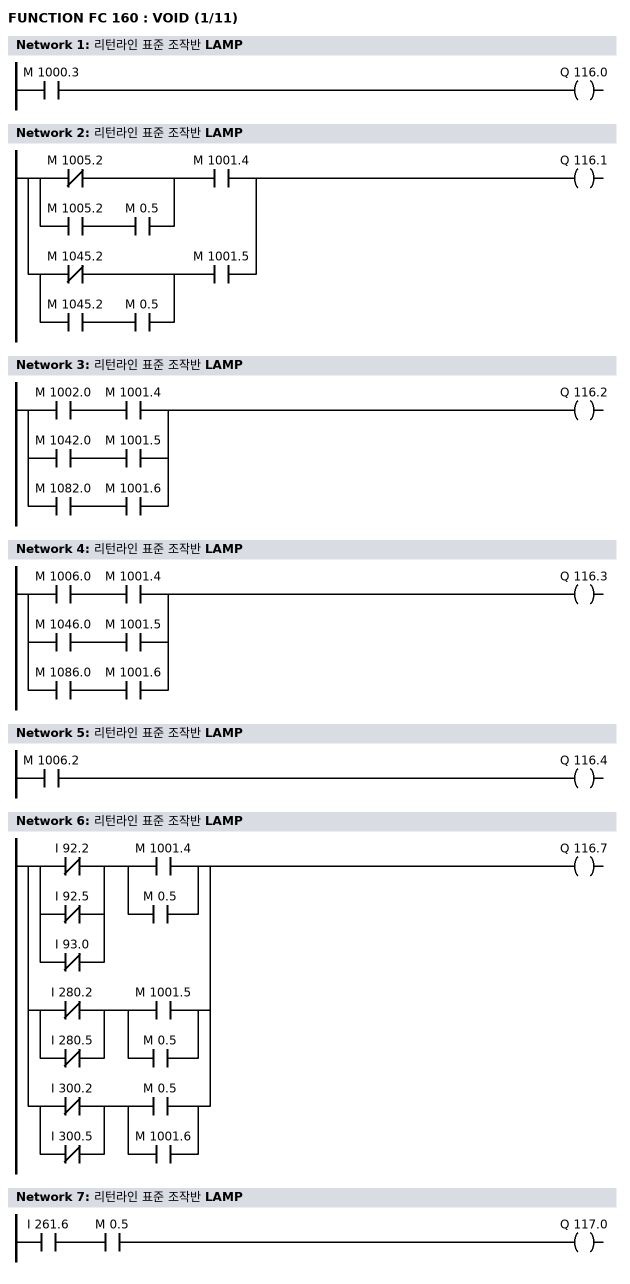

      A     M   1000.3;
      =     Q    116.0;
NETWORK
TITLE =리턴라인 표준 조작반 LAMP

      A(    ;
      ON    M   1005.2;
      O     ;
      A     M   1005.2;
      A     M      0.5;
      )     ;
      A     M   1001.4;
      O     ;
      A(    ;
      ON    M   1045.2;
      O     ;
      A     M   1045.2;
      A     M      0.5;
      )     ;
      A     M   1001.5;
      =     Q    116.1;
NETWORK
TITLE =리턴라인 표준 조작반 LAMP

      A     M   1002.0;
      A     M   1001.4;
      O     ;
      A     M   1042.0;
      A     M   1001.5;
      O     ;
      A     M   1082.0;
      A     M   1001.6;
      =     Q    116.2;
NETWORK
TITLE =리턴라인 표준 조작반 LAMP

      A     M   1006.0;
      A     M   1001.4;
      O     ;
      A     M   1046.0;
      A     M   1001.5;
      O     ;
      A     M   1086.0;
      A     M   1001.6;
      =     Q    116.3;
NETWORK
TITLE =리턴라인 표준 조작반 LAMP

      A     M   1006.2;
      =     Q    116.4;
NETWORK
TITLE =리턴라인 표준 조작반 LAMP

      A(    ;
      ON    I     92.2;
      ON    I     92.5;
      ON    I     93.0;
      )     ;
      A(    ;
      O     M   1001.4;
      O     M      0.5;
      )     ;
      O     ;
      A(    ;
      ON    I    280.2;
      ON    I    280.5;
      )     ;
      A(    ;
      O     M   1001.5;
      O     M      0.5;
      )     ;
      O     ;
      A(    ;
      ON    I    300.2;
      ON    I    300.5;
      )     ;
      A(    ;
      O     M      0.5;
      O     M   1001.6;
      )     ;
      =     Q    116.7;
NETWORK
TITLE =리턴라인 표준 조작반 LAMP

      A     I    261.6;
      A     M      0.5;
      =     Q    117.0;
NETWORK
TITLE =리턴라인 표준 조작반 LAMP
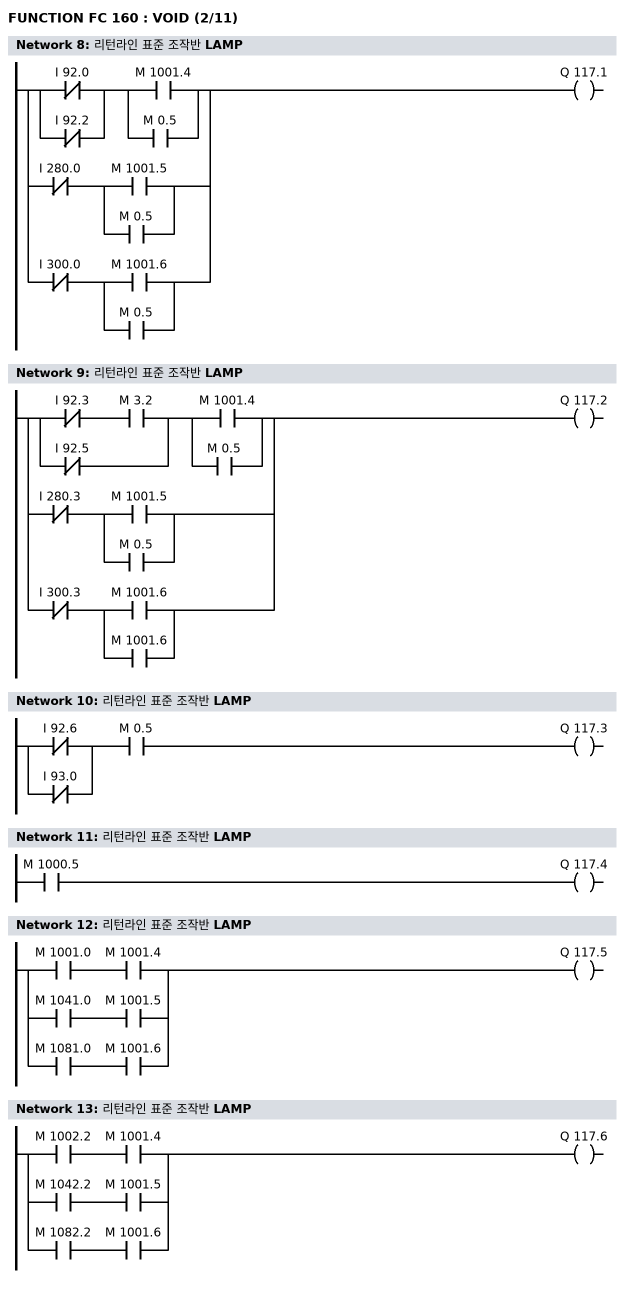

      A(    ;
      ON    I     92.0;
      ON    I     92.2;
      )     ;
      A(    ;
      O     M   1001.4;
      O     M      0.5;
      )     ;
      O     ;
      AN    I    280.0;
      A(    ;
      O     M   1001.5;
      O     M      0.5;
      )     ;
      O     ;
      AN    I    300.0;
      A(    ;
      O     M   1001.6;
      O     M      0.5;
      )     ;
      =     Q    117.1;
NETWORK
TITLE =리턴라인 표준 조작반 LAMP

      A(    ;
      AN    I     92.3;
      A     M      3.2;
      ON    I     92.5;
      )     ;
      A(    ;
      O     M   1001.4;
      O     M      0.5;
      )     ;
      O     ;
      AN    I    280.3;
      A(    ;
      O     M   1001.5;
      O     M      0.5;
      )     ;
      O     ;
      AN    I    300.3;
      A(    ;
      O     M   1001.6;
      O     M   1001.6;
      )     ;
      =     Q    117.2;
NETWORK
TITLE =리턴라인 표준 조작반 LAMP

      A(    ;
      ON    I     92.6;
      ON    I     93.0;
      )     ;
      A     M      0.5;
      =     Q    117.3;
NETWORK
TITLE =리턴라인 표준 조작반 LAMP

      A     M   1000.5;
      =     Q    117.4;
NETWORK
TITLE =리턴라인 표준 조작반 LAMP

      A     M   1001.0;
      A     M   1001.4;
      O     ;
      A     M   1041.0;
      A     M   1001.5;
      O     ;
      A     M   1081.0;
      A     M   1001.6;
      =     Q    117.5;
NETWORK
TITLE =리턴라인 표준 조작반 LAMP

      A     M   1002.2;
      A     M   1001.4;
      O     ;
      A     M   1042.2;
      A     M   1001.5;
      O     ;
      A     M   1082.2;
      A     M   1001.6;
      =     Q    117.6;
NETWORK
TITLE =리턴라인 표준 조작반 LAMP
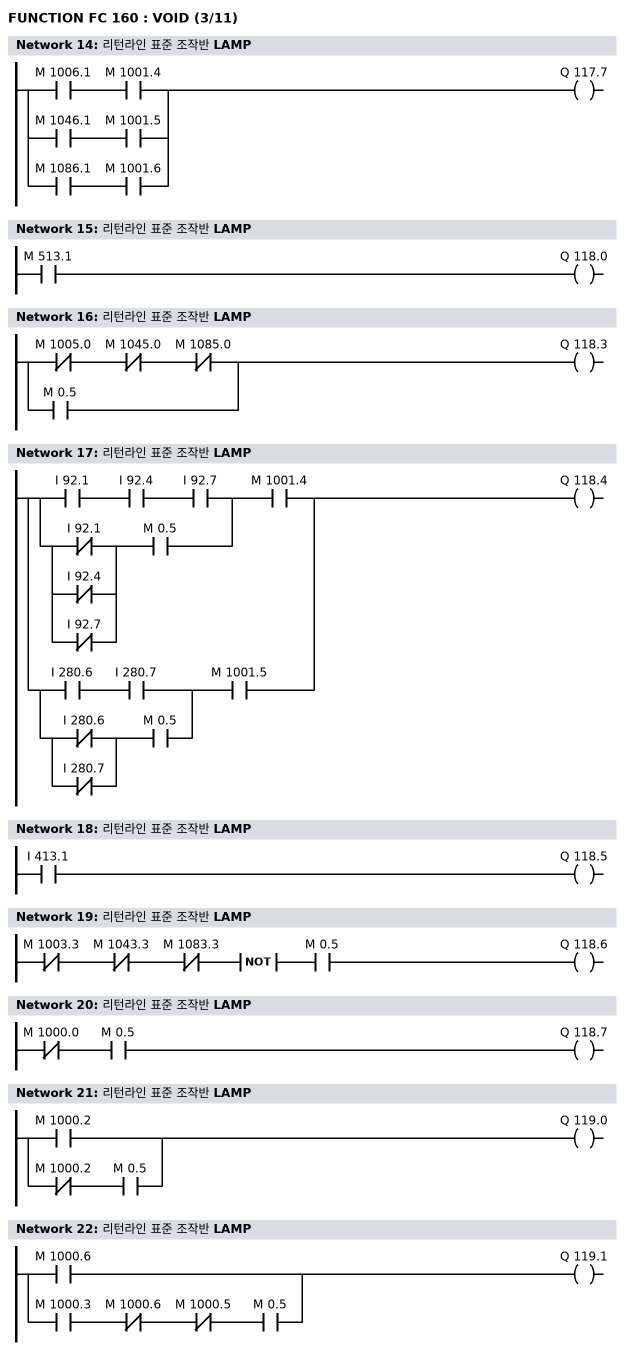

      A     M   1006.1;
      A     M   1001.4;
      O     ;
      A     M   1046.1;
      A     M   1001.5;
      O     ;
      A     M   1086.1;
      A     M   1001.6;
      =     Q    117.7;
NETWORK
TITLE =리턴라인 표준 조작반 LAMP

      A     M    513.1;
      =     Q    118.0;
NETWORK
TITLE =리턴라인 표준 조작반 LAMP

      AN    M   1005.0;
      AN    M   1045.0;
      AN    M   1085.0;
      O     M      0.5;
      =     Q    118.3;
NETWORK
TITLE =리턴라인 표준 조작반 LAMP

      A(    ;
      A     I     92.1;
      A     I     92.4;
      A     I     92.7;
      O     ;
      A(    ;
      ON    I     92.1;
      ON    I     92.4;
      ON    I     92.7;
      )     ;
      A     M      0.5;
      )     ;
      A     M   1001.4;
      O     ;
      A(    ;
      A     I    280.6;
      A     I    280.7;
      O     ;
      A(    ;
      ON    I    280.6;
      ON    I    280.7;
      )     ;
      A     M      0.5;
      )     ;
      A     M   1001.5;
      =     Q    118.4;
NETWORK
TITLE =리턴라인 표준 조작반 LAMP

      A     I    413.1;
      =     Q    118.5;
NETWORK
TITLE =리턴라인 표준 조작반 LAMP

      AN    M   1003.3;
      AN    M   1043.3;
      AN    M   1083.3;
      NOT   ;
      A     M      0.5;
      =     Q    118.6;
NETWORK
TITLE =리턴라인 표준 조작반 LAMP

      AN    M   1000.0;
      A     M      0.5;
      =     Q    118.7;
NETWORK
TITLE =리턴라인 표준 조작반 LAMP

      O     M   1000.2;
      O     ;
      AN    M   1000.2;
      A     M      0.5;
      =     Q    119.0;
NETWORK
TITLE =리턴라인 표준 조작반 LAMP

      O     M   1000.6;
      O     ;
      A     M   1000.3;
      AN    M   1000.6;
      AN    M   1000.5;
      A     M      0.5;
      =     Q    119.1;
NETWORK
TITLE =리턴라인 표준 조작반 LAMP
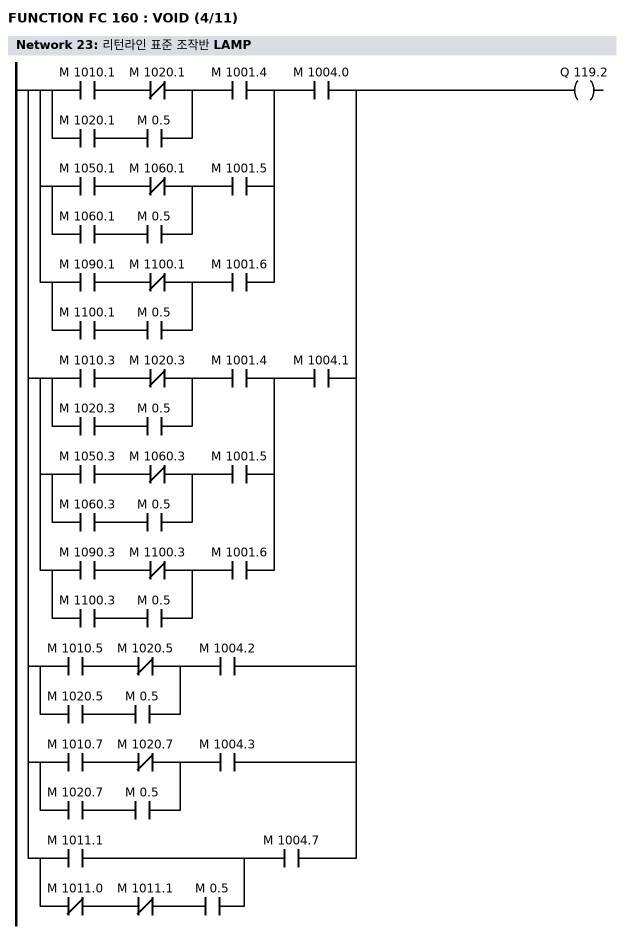

      A(    ;
      A(    ;
      A     M   1010.1;
      AN    M   1020.1;
      O     ;
      A     M   1020.1;
      A     M      0.5;
      )     ;
      A     M   1001.4;
      O     ;
      A(    ;
      A     M   1050.1;
      AN    M   1060.1;
      O     ;
      A     M   1060.1;
      A     M      0.5;
      )     ;
      A     M   1001.5;
      O     ;
      A(    ;
      A     M   1090.1;
      AN    M   1100.1;
      O     ;
      A     M   1100.1;
      A     M      0.5;
      )     ;
      A     M   1001.6;
      )     ;
      A     M   1004.0;
      O     ;
      A(    ;
      A(    ;
      A     M   1010.3;
      AN    M   1020.3;
      O     ;
      A     M   1020.3;
      A     M      0.5;
      )     ;
      A     M   1001.4;
      O     ;
      A(    ;
      A     M   1050.3;
      AN    M   1060.3;
      O     ;
      A     M   1060.3;
      A     M      0.5;
      )     ;
      A     M   1001.5;
      O     ;
      A(    ;
      A     M   1090.3;
      AN    M   1100.3;
      O     ;
      A     M   1100.3;
      A     M      0.5;
      )     ;
      A     M   1001.6;
      )     ;
      A     M   1004.1;
      O     ;
      A(    ;
      A     M   1010.5;
      AN    M   1020.5;
      O     ;
      A     M   1020.5;
      A     M      0.5;
      )     ;
      A     M   1004.2;
      O     ;
      A(    ;
      A     M   1010.7;
      AN    M   1020.7;
      O     ;
      A     M   1020.7;
      A     M      0.5;
      )     ;
      A     M   1004.3;
      O     ;
      A(    ;
      O     M   1011.1;
      O     ;
      AN    M   1011.0;
      AN    M   1011.1;
      A     M      0.5;
      )     ;
      A     M   1004.7;
      =     Q    119.2;
NETWORK
TITLE =리턴라인 표준 조작반 LAMP
